  MoveC 2623 to (57.81, -73.19, -4) mm, rotated rx 180 ry 0 rz 90 deg; joints [72.07, -16.046, 78.681, 0, 27.365, 72.07] to (57.8, -69.17, -4) mm, rotated rx 180 ry 0 rz 90 deg; joints [72.193, -16.074, 78.779, 0, 27.295, 72.193]
  MoveL 2624 to (57.48, -68.7, -4) mm, rotated rx -180 ry 0 rz 90 deg; joints [72.204, -16.085, 78.814, 0, 27.271, 72.204]
  MoveL 2625 to (54.49, -65.17, -4) mm, rotated rx 180 ry 0 rz 90 deg; joints [72.283, -16.175, 79.122, 0, 27.052, 72.283]
  MoveL 2626 to (28.89, -35.54, -4) mm, rotated rx -180 ry 0 rz 90 deg; joints [72.956, -16.906, 81.694, 0, 25.212, 72.956]
  MoveL 2627 to (27.54, -34.02, -4) mm, rotated rx 180 ry 0 rz 90 deg; joints [72.991, -16.943, 81.826, 0, 25.117, 72.991]
  MoveL 2628 to (13.23, -22.57, -4) mm, rotated rx 180 ry 0 rz 90 deg; joints [73.216, -17.293, 83.111, 0, 24.182, 73.216]
  MoveC 2629 to (12.1, -21.76, -4) mm, rotated rx -180 ry 0 rz 90 deg; joints [73.231, -17.319, 83.209, 0, 24.11, 73.231] to (10.9, -21.09, -4) mm, rotated rx 180 ry 0 rz 90 deg; joints [73.241, -17.346, 83.31, 0, 24.036, 73.241]
  MoveC 2630 to (6.62, -20.99, -4) mm, rotated rx 180 ry 0 rz 90 deg; joints [73.203, -17.429, 83.618, 0, 23.81, 73.203] to (3.75, -24.17, -4) mm, rotated rx 180 ry 0 rz 90 deg; joints [73.074, -17.465, 83.754, 0, 23.711, 73.074]
  MoveL 2631 to (3.46, -25.11, -4) mm, rotated rx -180 ry 0 rz 90 deg; joints [73.04, -17.465, 83.754, 0, 23.711, 73.04]
  MoveL 2632 to (-7.61, -66.81, -4) mm, rotated rx 180 ry 0 rz 90 deg; joints [71.6, -17.423, 83.597, 0, 23.826, 71.6]
  MoveL 2633 to (-8.62, -70.6, -4) mm, rotated rx 180 ry 0 rz 90 deg; joints [71.469, -17.418, 83.578, 0, 23.84, 71.469]
  MoveL 2634 to (-8.77, -71.55, -4) mm, rotated rx -180 ry 0 rz 90 deg; joints [71.437, -17.415, 83.566, 0, 23.849, 71.437]
  MoveC 2635 to (-8.03, -75.01, -4) mm, rotated rx 180 ry 0 rz 90 deg; joints [71.336, -17.379, 83.432, 0, 23.947, 71.336] to (-5.21, -77.15, -4) mm, rotated rx 180 ry 0 rz 90 deg; joints [71.298, -17.312, 83.181, 0, 24.131, 71.298]
  MoveC 2636 to (-3.81, -77.46, -4) mm, rotated rx -180 ry 0 rz 90 deg; joints [71.303, -17.283, 83.073, 0, 24.21, 71.303] to (-2.37, -77.54, -4) mm, rotated rx -180 ry 0 rz 90 deg; joints [71.316, -17.255, 82.969, 0, 24.286, 71.316]
  MoveL 2637 to (25.78, -77.25, -4) mm, rotated rx 180 ry 0 rz 90 deg; joints [71.62, -16.698, 80.95, 0, 25.748, 71.62]
  MoveL 2638 to (25.7, -69.7, -4) mm, rotated rx 180 ry 0 rz 90 deg; joints [71.855, -16.751, 81.137, 0, 25.614, 71.855]
  MoveL 2639 to (25.7, -69.7, -1) mm, rotated rx 180 ry 0 rz 90 deg; joints [71.855, -16.902, 81.239, 0, 25.664, 71.855]
  Establecer velocidad (1000.0 mm/s)
  MoveL 2640 to (25.7, -69.7, 10) mm, rotated rx 180 ry 0 rz 90 deg; joints [71.855, -17.457, 81.607, 0, 25.851, 71.855]
  Establecer velocidad (66.7 mm/s)
  MoveL 2641 to (67.55, -30.93, 10) mm, rotated rx -180 ry 0 rz 90 deg; joints [73.464, -16.821, 79.406, 0, 27.415, 73.464]
  MoveL 2642 to (67.55, -30.93, -0.75) mm, rotated rx -180 ry 0 rz 90 deg; joints [73.464, -16.283, 79.045, 0, 27.238, 73.464]
  MoveL 2643 to (69.05, -31.11, -1.16) mm, rotated rx -180 ry 0 rz 90 deg; joints [73.472, -16.228, 78.914, 0, 27.314, 73.472]
  MoveL 2644 to (70.56, -30.93, -1.56) mm, rotated rx 180 ry 0 rz 90 deg; joints [73.492, -16.176, 78.79, 0, 27.385, 73.492]
  MoveL 2645 to (71.99, -30.42, -1.97) mm, rotated rx -180 ry 0 rz 90 deg; joints [73.521, -16.127, 78.68, 0, 27.447, 73.521]
  MoveL 2646 to (73.27, -29.6, -2.37) mm, rotated rx 180 ry 0 rz 90 deg; joints [73.558, -16.083, 78.587, 0, 27.496, 73.558]
  MoveL 2647 to (74.34, -28.52, -2.78) mm, rotated rx -180 ry 0 rz 90 deg; joints [73.601, -16.046, 78.516, 0, 27.53, 73.601]
  MoveL 2648 to (75.15, -27.24, -3.19) mm, rotated rx 180 ry 0 rz 90 deg; joints [73.648, -16.016, 78.47, 0, 27.546, 73.648]
  MoveL 2649 to (75.65, -25.8, -3.59) mm, rotated rx -180 ry 0 rz 90 deg; joints [73.696, -15.994, 78.45, 0, 27.544, 73.696]
  MoveL 2650 to (75.78, -24.29, -4) mm, rotated rx -180 ry 0 rz 90 deg; joints [73.744, -15.98, 78.46, 0, 27.521, 73.744]
  MoveL 2651 to (75.78, -5.21, -4) mm, rotated rx -180 ry 0 rz 90 deg; joints [74.335, -16.102, 78.873, 0, 27.229, 74.335]
  MoveL 2652 to (75.77, -4.51, -4) mm, rotated rx 180 ry 0 rz 90 deg; joints [74.357, -16.107, 78.889, 0, 27.217, 74.357]
  MoveC 2653 to (73.31, -1.48, -4) mm, rotated rx -180 ry 0 rz 90 deg; joints [74.43, -16.18, 79.139, 0, 27.041, 74.43] to (69.65, -0.12, -4) mm, rotated rx -180 ry 0 rz 90 deg; joints [74.44, -16.268, 79.443, 0, 26.825, 74.44]
  MoveC 2654 to (68.39, -0.22, -4) mm, rotated rx 180 ry 0 rz 90 deg; joints [74.426, -16.295, 79.536, 0, 26.759, 74.426] to (67.21, -0.66, -4) mm, rotated rx -180 ry 0 rz 90 deg; joints [74.402, -16.318, 79.615, 0, 26.702, 74.402]
  MoveL 2655 to (66.63, -1.42, -4) mm, rotated rx 180 ry 0 rz 90 deg; joints [74.373, -16.326, 79.643, 0, 26.683, 74.373]
  MoveL 2656 to (51.65, -21.98, -4) mm, rotated rx 180 ry 0 rz 90 deg; joints [73.596, -16.52, 80.321, 0, 26.199, 73.596]
  MoveL 2657 to (50.74, -23.24, -4) mm, rotated rx 180 ry 0 rz 90 deg; joints [73.549, -16.531, 80.36, 0, 26.171, 73.549]
  MoveC 2658 to (49.85, -26.2, -4) mm, rotated rx 180 ry 0 rz 90 deg; joints [73.448, -16.532, 80.361, 0, 26.17, 73.448] to (50.96, -29.09, -4) mm, rotated rx -180 ry 0 rz 90 deg; joints [73.368, -16.49, 80.215, 0, 26.275, 73.368]
  MoveL 2659 to (51.59, -29.85, -4) mm, rotated rx -180 ry 0 rz 90 deg; joints [73.35, -16.472, 80.151, 0, 26.32, 73.35]
  MoveL 2660 to (67.24, -47.54, -4) mm, rotated rx 180 ry 0 rz 90 deg; joints [72.949, -16.016, 78.579, 0, 27.436, 72.949]
  MoveL 2661 to (67.55, -47.86, -4) mm, rotated rx -180 ry 0 rz 90 deg; joints [72.942, -16.007, 78.549, 0, 27.458, 72.942]
  MoveC 2662 to (68.55, -48.33, -4) mm, rotated rx -180 ry 0 rz 90 deg; joints [72.937, -15.981, 78.463, 0, 27.519, 72.937] to (69.65, -48.44, -4) mm, rotated rx -180 ry 0 rz 90 deg; joints [72.944, -15.956, 78.377, 0, 27.579, 72.944]
  MoveC 2663 to (73.34, -47.15, -4) mm, rotated rx 180 ry 0 rz 90 deg; joints [73.018, -15.882, 78.127, 0, 27.755, 73.018] to (75.75, -44.07, -4) mm, rotated rx -180 ry 0 rz 90 deg; joints [73.135, -15.849, 78.016, 0, 27.833, 73.135]
  MoveL 2664 to (75.79, -43.12, -4) mm, rotated rx 180 ry 0 rz 90 deg; joints [73.165, -15.855, 78.034, 0, 27.82, 73.165]
  MoveL 2665 to (75.78, -24.29, -4) mm, rotated rx -180 ry 0 rz 90 deg; joints [73.744, -15.98, 78.46, 0, 27.521, 73.744]
  MoveL 2666 to (68.23, -24.29, -4) mm, rotated rx 180 ry 0 rz 90 deg; joints [73.676, -16.148, 79.03, 0, 27.118, 73.676]
  MoveL 2667 to (68.23, -24.29, -1) mm, rotated rx -180 ry 0 rz 90 deg; joints [73.676, -16.298, 79.132, 0, 27.166, 73.676]
  Establecer velocidad (1000.0 mm/s)
  MoveL 2668 to (68.23, -24.29, 10) mm, rotated rx 180 ry 0 rz 90 deg; joints [73.676, -16.849, 79.502, 0, 27.348, 73.676]
  Establecer velocidad (66.7 mm/s)
  MoveL 2669 to (36.34, 8.62, 10) mm, rotated rx 180 ry 0 rz 90 deg; joints [74.423, -17.725, 82.561, 0, 25.164, 74.423]
  MoveL 2670 to (36.34, 8.62, -0.75) mm, rotated rx 180 ry 0 rz 90 deg; joints [74.423, -17.181, 82.202, 0, 24.979, 74.423]
  MoveL 2671 to (37.46, 7.59, -1.16) mm, rotated rx 180 ry 0 rz 90 deg; joints [74.4, -17.132, 82.086, 0, 25.046, 74.4]
  MoveL 2672 to (38.79, 6.86, -1.56) mm, rotated rx -180 ry 0 rz 90 deg; joints [74.389, -17.08, 81.96, 0, 25.12, 74.389]
  MoveL 2673 to (40.25, 6.44, -1.97) mm, rotated rx 180 ry 0 rz 90 deg; joints [74.389, -17.028, 81.831, 0, 25.197, 74.389]
  MoveL 2674 to (41.77, 6.36, -2.37) mm, rotated rx -180 ry 0 rz 90 deg; joints [74.399, -16.976, 81.704, 0, 25.272, 74.399]
  MoveL 2675 to (43.27, 6.61, -2.78) mm, rotated rx 180 ry 0 rz 90 deg; joints [74.421, -16.926, 81.585, 0, 25.341, 74.421]
  MoveL 2676 to (44.68, 7.19, -3.19) mm, rotated rx 180 ry 0 rz 90 deg; joints [74.452, -16.88, 81.48, 0, 25.4, 74.452]
  MoveL 2677 to (45.92, 8.07, -3.59) mm, rotated rx 180 ry 0 rz 90 deg; joints [74.49, -16.839, 81.393, 0, 25.446, 74.49]
  MoveL 2678 to (46.91, 9.21, -4) mm, rotated rx 180 ry 0 rz 90 deg; joints [74.535, -16.805, 81.329, 0, 25.475, 74.535]
  MoveL 2679 to (58.63, 25.57, -4) mm, rotated rx 180 ry 0 rz 90 deg; joints [75.153, -16.653, 80.79, 0, 25.864, 75.153]
  MoveC 2680 to (58.89, 26.03, -4) mm, rotated rx 180 ry 0 rz 90 deg; joints [75.17, -16.65, 80.779, 0, 25.871, 75.17] to (59.04, 26.54, -4) mm, rotated rx 180 ry 0 rz 90 deg; joints [75.187, -16.65, 80.778, 0, 25.872, 75.187]
  MoveC 2681 to (58.64, 30.12, -4) mm, rotated rx 180 ry 0 rz 90 deg; joints [75.297, -16.678, 80.878, 0, 25.8, 75.297] to (56.35, 32.91, -4) mm, rotated rx -180 ry 0 rz 90 deg; joints [75.366, -16.741, 81.102, 0, 25.639, 75.366]
  MoveC 2682 to (55.39, 33.36, -4) mm, rotated rx -180 ry 0 rz 90 deg; joints [75.373, -16.764, 81.183, 0, 25.581, 75.373] to (54.33, 33.5, -4) mm, rotated rx -180 ry 0 rz 90 deg; joints [75.368, -16.786, 81.264, 0, 25.523, 75.368]
  MoveL 2683 to (46.91, 33.32, -4) mm, rotated rx -180 ry 0 rz 90 deg; joints [75.301, -16.938, 81.808, 0, 25.13, 75.301]
  MoveL 2684 to (7.5, 32.25, -4) mm, rotated rx 180 ry 0 rz 90 deg; joints [74.929, -17.696, 84.638, 0, 23.058, 74.929]
  MoveC 2685 to (4.94, 31.58, -4) mm, rotated rx -180 ry 0 rz 90 deg; joints [74.885, -17.74, 84.808, 0, 22.932, 74.885] to (2.93, 29.85, -4) mm, rotated rx -180 ry 0 rz 90 deg; joints [74.811, -17.768, 84.917, 0, 22.852, 74.811]
  MoveC 2686 to (2.15, 27.7, -4) mm, rotated rx 180 ry 0 rz 90 deg; joints [74.734, -17.772, 84.931, 0, 22.841, 74.734] to (2.37, 25.41, -4) mm, rotated rx -180 ry 0 rz 90 deg; joints [74.661, -17.757, 84.871, 0, 22.886, 74.661]
  MoveL 2687 to (2.79, 24.17, -4) mm, rotated rx -180 ry 0 rz 90 deg; joints [74.625, -17.743, 84.817, 0, 22.926, 74.625]
  MoveL 2688 to (8.64, 8.05, -4) mm, rotated rx -180 ry 0 rz 90 deg; joints [74.155, -17.551, 84.08, 0, 23.47, 74.155]
  MoveC 2689 to (9.35, 6.7, -4) mm, rotated rx -180 ry 0 rz 90 deg; joints [74.118, -17.53, 84.002, 0, 23.528, 74.118] to (10.39, 5.59, -4) mm, rotated rx 180 ry 0 rz 90 deg; joints [74.092, -17.505, 83.906, 0, 23.599, 74.092]
  MoveL 2690 to (27.01, -7.35, -4) mm, rotated rx 180 ry 0 rz 90 deg; joints [73.831, -17.112, 82.441, 0, 24.67, 73.831]
  MoveL 2691 to (27.96, -8.06, -4) mm, rotated rx -180 ry 0 rz 90 deg; joints [73.817, -17.089, 82.358, 0, 24.731, 73.817]
  MoveC 2692 to (31.75, -9.06, -4) mm, rotated rx -180 ry 0 rz 90 deg; joints [73.82, -17.007, 82.061, 0, 24.946, 73.82] to (35.15, -7.11, -4) mm, rotated rx 180 ry 0 rz 90 deg; joints [73.913, -16.95, 81.854, 0, 25.096, 73.913]
  MoveL 2693 to (35.89, -6.16, -4) mm, rotated rx 180 ry 0 rz 90 deg; joints [73.95, -16.941, 81.82, 0, 25.121, 73.95]
  MoveL 2694 to (46.91, 9.21, -4) mm, rotated rx 180 ry 0 rz 90 deg; joints [74.535, -16.805, 81.329, 0, 25.475, 74.535]
  MoveL 2695 to (40.77, 13.61, -4) mm, rotated rx -180 ry 0 rz 90 deg; joints [74.621, -16.955, 81.87, 0, 25.085, 74.621]
  MoveL 2696 to (40.77, 13.61, -1) mm, rotated rx 180 ry 0 rz 90 deg; joints [74.621, -17.107, 81.971, 0, 25.136, 74.621]
  Establecer velocidad (1000.0 mm/s)
  MoveL 2697 to (40.77, 13.61, 10) mm, rotated rx 180 ry 0 rz 90 deg; joints [74.621, -17.663, 82.338, 0, 25.325, 74.621]
  Establecer velocidad (66.7 mm/s)
  MoveL 2698 to (26.76, 68.82, 10) mm, rotated rx -180 ry 0 rz 90 deg; joints [76.28, -18.225, 84.399, 0, 23.827, 76.28]
  MoveL 2699 to (26.76, 68.82, -0.75) mm, rotated rx -180 ry 0 rz 90 deg; joints [76.28, -17.677, 84.041, 0, 23.637, 76.28]
  MoveL 2700 to (26.96, 70.32, -1.16) mm, rotated rx 180 ry 0 rz 90 deg; joints [76.331, -17.66, 84.039, 0, 23.621, 76.331]
  MoveL 2701 to (26.79, 71.84, -1.56) mm, rotated rx 180 ry 0 rz 90 deg; joints [76.379, -17.649, 84.064, 0, 23.585, 76.379]
  MoveL 2702 to (26.29, 73.27, -1.97) mm, rotated rx 180 ry 0 rz 90 deg; joints [76.422, -17.645, 84.111, 0, 23.534, 76.422]
  MoveL 2703 to (25.49, 74.56, -2.37) mm, rotated rx 180 ry 0 rz 90 deg; joints [76.457, -17.645, 84.177, 0, 23.467, 76.457]
  MoveL 2704 to (24.42, 75.64, -2.78) mm, rotated rx 180 ry 0 rz 90 deg; joints [76.484, -17.649, 84.259, 0, 23.39, 76.484]
  MoveL 2705 to (23.14, 76.46, -3.19) mm, rotated rx 180 ry 0 rz 90 deg; joints [76.501, -17.656, 84.352, 0, 23.304, 76.501]
  MoveL 2706 to (21.71, 76.98, -3.59) mm, rotated rx -180 ry 0 rz 90 deg; joints [76.506, -17.665, 84.45, 0, 23.215, 76.506]
  MoveL 2707 to (20.21, 77.13, -4) mm, rotated rx -180 ry 0 rz 90 deg; joints [76.5, -17.673, 84.547, 0, 23.126, 76.5]
  MoveL 2708 to (-28.9, 77.66, -4) mm, rotated rx -180 ry 0 rz 90 deg; joints [76.12, -18.533, 88.011, 0, 20.522, 76.12]
  MoveL 2709 to (-30.61, 77.66, -4) mm, rotated rx -180 ry 0 rz 90 deg; joints [76.106, -18.561, 88.129, 0, 20.432, 76.106]
  MoveC 2710 to (-32.6, 77.56, -4) mm, rotated rx -180 ry 0 rz 90 deg; joints [76.086, -18.593, 88.264, 0, 20.329, 76.086] to (-34.56, 77.23, -4) mm, rotated rx 180 ry 0 rz 90 deg; joints [76.059, -18.623, 88.394, 0, 20.23, 76.059]
  MoveC 2711 to (-37.55, 73.36, -4) mm, rotated rx 180 ry 0 rz 90 deg; joints [75.903, -18.656, 88.533, 0, 20.123, 75.903] to (-36.68, 68.53, -4) mm, rotated rx 180 ry 0 rz 90 deg; joints [75.748, -18.622, 88.389, 0, 20.233, 75.748]
  MoveC 2712 to (-34.85, 67.27, -4) mm, rotated rx 180 ry 0 rz 90 deg; joints [75.721, -18.588, 88.242, 0, 20.346, 75.721] to (-32.99, 66.06, -4) mm, rotated rx -180 ry 0 rz 90 deg; joints [75.696, -18.553, 88.092, 0, 20.46, 75.696]
  MoveL 2713 to (-12.79, 53.26, -4) mm, rotated rx 180 ry 0 rz 90 deg; joints [75.443, -18.159, 86.463, 0, 21.696, 75.443]
  MoveL 2714 to (-11.85, 52.68, -4) mm, rotated rx 180 ry 0 rz 90 deg; joints [75.431, -18.14, 86.386, 0, 21.754, 75.431]
  MoveC 2715 to (-9.56, 51.76, -4) mm, rotated rx -180 ry 0 rz 90 deg; joints [75.421, -18.096, 86.209, 0, 21.887, 75.421] to (-7.11, 51.53, -4) mm, rotated rx -180 ry 0 rz 90 deg; joints [75.434, -18.052, 86.032, 0, 22.019, 75.434]
  MoveL 2716 to (70.6, 57.18, -4) mm, rotated rx 180 ry 0 rz 90 deg; joints [76.25, -16.57, 80.498, 0, 26.073, 76.25]
  MoveL 2717 to (71.37, 57.27, -4) mm, rotated rx 180 ry 0 rz 90 deg; joints [76.259, -16.554, 80.441, 0, 26.113, 76.259]
  MoveC 2718 to (74.16, 58.71, -4) mm, rotated rx 180 ry 0 rz 90 deg; joints [76.327, -16.502, 80.258, 0, 26.244, 76.327] to (75.32, 61.63, -4) mm, rotated rx -180 ry 0 rz 90 deg; joints [76.428, -16.493, 80.225, 0, 26.268, 76.428]
  MoveL 2719 to (75.32, 62.07, -4) mm, rotated rx 180 ry 0 rz 90 deg; joints [76.442, -16.495, 80.232, 0, 26.263, 76.442]
  MoveL 2720 to (75.32, 71.55, -4) mm, rotated rx -180 ry 0 rz 90 deg; joints [76.742, -16.543, 80.402, 0, 26.141, 76.742]
  MoveL 2721 to (75.31, 71.95, -4) mm, rotated rx -180 ry 0 rz 90 deg; joints [76.755, -16.546, 80.411, 0, 26.135, 76.755]
  MoveC 2722 to (74, 74.91, -4) mm, rotated rx 180 ry 0 rz 90 deg; joints [76.839, -16.588, 80.561, 0, 26.027, 76.839] to (71.02, 76.18, -4) mm, rotated rx -180 ry 0 rz 90 deg; joints [76.858, -16.658, 80.807, 0, 25.851, 76.858]
  MoveC 2723 to (46.95, 76.74, -4) mm, rotated rx 180 ry 0 rz 90 deg; joints [76.694, -17.155, 82.6, 0, 24.555, 76.694] to (22.88, 77.1, -4) mm, rotated rx -180 ry 0 rz 90 deg; joints [76.52, -17.623, 84.355, 0, 23.268, 76.52]
  MoveL 2724 to (20.21, 77.13, -4) mm, rotated rx -180 ry 0 rz 90 deg; joints [76.5, -17.673, 84.547, 0, 23.126, 76.5]
  MoveL 2725 to (20.12, 69.58, -4) mm, rotated rx -180 ry 0 rz 90 deg; joints [76.252, -17.64, 84.422, 0, 23.218, 76.252]
  MoveL 2726 to (20.12, 69.58, -1) mm, rotated rx 180 ry 0 rz 90 deg; joints [76.252, -17.793, 84.523, 0, 23.271, 76.252]
  Establecer velocidad (1000.0 mm/s)
  MoveL 2727 to (20.12, 69.58, 10) mm, rotated rx -180 ry 0 rz 90 deg; joints [76.252, -18.355, 84.889, 0, 23.466, 76.252]
  Establecer velocidad (66.7 mm/s)
  MoveL 2728 to (26.76, 68.55, 10) mm, rotated rx 180 ry 0 rz 90 deg; joints [76.271, -18.224, 84.394, 0, 23.83, 76.271]
  MoveL 2729 to (26.76, 68.55, -1) mm, rotated rx -180 ry 0 rz 90 deg; joints [76.271, -17.663, 84.027, 0, 23.636, 76.271]
  MoveL 2730 to (26.96, 70.05, -1.41) mm, rotated rx 180 ry 0 rz 90 deg; joints [76.322, -17.646, 84.026, 0, 23.62, 76.322]
  MoveL 2731 to (26.79, 71.56, -1.81) mm, rotated rx 180 ry 0 rz 90 deg; joints [76.37, -17.635, 84.05, 0, 23.585, 76.37]
  MoveL 2732 to (26.29, 73, -2.22) mm, rotated rx 180 ry 0 rz 90 deg; joints [76.413, -17.63, 84.098, 0, 23.533, 76.413]
  MoveL 2733 to (25.49, 74.29, -2.62) mm, rotated rx 180 ry 0 rz 90 deg; joints [76.448, -17.631, 84.164, 0, 23.467, 76.448]
  MoveL 2734 to (24.42, 75.37, -3.03) mm, rotated rx -180 ry 0 rz 90 deg; joints [76.475, -17.635, 84.247, 0, 23.389, 76.475]
  MoveL 2735 to (23.14, 76.19, -3.44) mm, rotated rx 180 ry 0 rz 90 deg; joints [76.492, -17.642, 84.339, 0, 23.303, 76.492]
  MoveL 2736 to (21.71, 76.7, -3.84) mm, rotated rx 180 ry 0 rz 90 deg; joints [76.497, -17.651, 84.437, 0, 23.214, 76.497]
  MoveL 2737 to (20.2, 76.86, -4.25) mm, rotated rx 180 ry 0 rz 90 deg; joints [76.491, -17.659, 84.534, 0, 23.125, 76.491]
  MoveC 2738 to (19.81, 76.86, -4.25) mm, rotated rx 180 ry 0 rz 90 deg; joints [76.488, -17.666, 84.562, 0, 23.104, 76.488] to (19.43, 76.86, -4.25) mm, rotated rx -180 ry 0 rz 90 deg; joints [76.485, -17.673, 84.59, 0, 23.083, 76.485]
  MoveL 2739 to (-29.85, 77.36, -4.25) mm, rotated rx -180 ry 0 rz 90 deg; joints [76.102, -18.535, 88.063, 0, 20.472, 76.102]
  MoveC 2740 to (-31.85, 77.3, -4.25) mm, rotated rx -180 ry 0 rz 90 deg; joints [76.084, -18.567, 88.2, 0, 20.367, 76.084] to (-33.83, 77.08, -4.25) mm, rotated rx 180 ry 0 rz 90 deg; joints [76.06, -18.598, 88.333, 0, 20.266, 76.06]
  MoveC 2741 to (-36.86, 73.32, -4.25) mm, rotated rx -180 ry 0 rz 90 deg; joints [75.907, -18.632, 88.476, 0, 20.156, 75.907] to (-36.19, 68.55, -4.25) mm, rotated rx 180 ry 0 rz 90 deg; joints [75.752, -18.602, 88.347, 0, 20.254, 75.752]
  MoveL 2742 to (-34.59, 67.43, -4.25) mm, rotated rx 180 ry 0 rz 90 deg; joints [75.728, -18.571, 88.218, 0, 20.353, 75.728]
  MoveL 2743 to (-27.63, 63.02, -4.25) mm, rotated rx -180 ry 0 rz 90 deg; joints [75.64, -18.439, 87.661, 0, 20.778, 75.64]
  MoveL 2744 to (-11.99, 53.11, -4.25) mm, rotated rx 180 ry 0 rz 90 deg; joints [75.444, -18.131, 86.395, 0, 21.736, 75.444]
  MoveC 2745 to (-9.54, 52.06, -4.25) mm, rotated rx 180 ry 0 rz 90 deg; joints [75.431, -18.084, 86.204, 0, 21.88, 75.431] to (-6.89, 51.83, -4.25) mm, rotated rx 180 ry 0 rz 90 deg; joints [75.446, -18.036, 86.014, 0, 22.022, 75.446]
  MoveC 2746 to (28.54, 54.43, -4.25) mm, rotated rx 180 ry 0 rz 90 deg; joints [75.827, -17.396, 83.536, 0, 23.86, 75.827] to (63.97, 57, -4.25) mm, rotated rx 180 ry 0 rz 90 deg; joints [76.193, -16.697, 80.982, 0, 25.715, 76.193]
  MoveL 2747 to (70.93, 57.56, -4.25) mm, rotated rx 180 ry 0 rz 90 deg; joints [76.265, -16.553, 80.471, 0, 26.082, 76.265]
  MoveC 2748 to (73.83, 58.97, -4.25) mm, rotated rx 180 ry 0 rz 90 deg; joints [76.332, -16.498, 80.28, 0, 26.219, 76.332] to (75, 61.98, -4.25) mm, rotated rx -180 ry 0 rz 90 deg; joints [76.436, -16.489, 80.246, 0, 26.243, 76.436]
  MoveL 2749 to (75, 71.52, -4.25) mm, rotated rx -180 ry 0 rz 90 deg; joints [76.739, -16.537, 80.417, 0, 26.12, 76.739]
  MoveC 2750 to (73.78, 74.54, -4.25) mm, rotated rx -180 ry 0 rz 90 deg; joints [76.826, -16.579, 80.563, 0, 26.016, 76.826] to (70.79, 75.86, -4.25) mm, rotated rx -180 ry 0 rz 90 deg; joints [76.845, -16.649, 80.81, 0, 25.839, 76.845]
  MoveC 2751 to (45.5, 76.48, -4.25) mm, rotated rx -180 ry 0 rz 90 deg; joints [76.674, -17.17, 82.694, 0, 24.476, 76.674] to (20.2, 76.86, -4.25) mm, rotated rx 180 ry 0 rz 90 deg; joints [76.491, -17.659, 84.534, 0, 23.125, 76.491]
  MoveL 2752 to (20.12, 69.31, -4.25) mm, rotated rx -180 ry 0 rz 90 deg; joints [76.243, -17.626, 84.409, 0, 23.218, 76.243]
  MoveL 2753 to (20.12, 69.31, -1.25) mm, rotated rx 180 ry 0 rz 90 deg; joints [76.243, -17.779, 84.51, 0, 23.27, 76.243]
  Establecer velocidad (1000.0 mm/s)
  MoveL 2754 to (20.12, 69.31, 10) mm, rotated rx 180 ry 0 rz 90 deg; joints [76.243, -18.354, 84.884, 0, 23.47, 76.243]
  Establecer velocidad (66.7 mm/s)
  MoveL 2755 to (37.85, 24.53, 10) mm, rotated rx 180 ry 0 rz 90 deg; joints [74.944, -17.783, 82.769, 0, 25.013, 74.944]
  MoveL 2756 to (37.85, 24.53, -1) mm, rotated rx -180 ry 0 rz 90 deg; joints [74.944, -17.225, 82.402, 0, 24.823, 74.944]
  MoveL 2757 to (38, 26.04, -1.41) mm, rotated rx 180 ry 0 rz 90 deg; joints [74.993, -17.21, 82.407, 0, 24.803, 74.993]
  MoveL 2758 to (37.77, 27.54, -1.81) mm, rotated rx 180 ry 0 rz 90 deg; joints [75.039, -17.202, 82.439, 0, 24.763, 75.039]
  MoveL 2759 to (37.22, 28.96, -2.22) mm, rotated rx 180 ry 0 rz 90 deg; joints [75.08, -17.2, 82.493, 0, 24.706, 75.08]
  MoveL 2760 to (36.37, 30.22, -2.62) mm, rotated rx -180 ry 0 rz 90 deg; joints [75.113, -17.203, 82.566, 0, 24.637, 75.113]
  MoveL 2761 to (35.26, 31.26, -3.03) mm, rotated rx -180 ry 0 rz 90 deg; joints [75.137, -17.21, 82.653, 0, 24.556, 75.137]
  MoveL 2762 to (33.95, 32.03, -3.44) mm, rotated rx 180 ry 0 rz 90 deg; joints [75.15, -17.219, 82.75, 0, 24.469, 75.15]
  MoveL 2763 to (32.5, 32.49, -3.84) mm, rotated rx -180 ry 0 rz 90 deg; joints [75.153, -17.229, 82.85, 0, 24.379, 75.153]
  MoveL 2764 to (30.99, 32.59, -4.25) mm, rotated rx 180 ry 0 rz 90 deg; joints [75.143, -17.239, 82.948, 0, 24.29, 75.143]
  MoveL 2765 to (8.05, 31.96, -4.25) mm, rotated rx 180 ry 0 rz 90 deg; joints [74.925, -17.672, 84.585, 0, 23.087, 74.925]
  MoveL 2766 to (7.11, 31.9, -4.25) mm, rotated rx 180 ry 0 rz 90 deg; joints [74.914, -17.689, 84.651, 0, 23.038, 74.914]
  MoveC 2767 to (3.22, 29.6, -4.25) mm, rotated rx -180 ry 0 rz 90 deg; joints [74.805, -17.749, 84.884, 0, 22.866, 74.805] to (2.78, 25.11, -4.25) mm, rotated rx 180 ry 0 rz 90 deg; joints [74.655, -17.735, 84.828, 0, 22.907, 74.655]
  MoveL 2768 to (8.98, 8.05, -4.25) mm, rotated rx -180 ry 0 rz 90 deg; joints [74.159, -17.532, 84.048, 0, 23.484, 74.159]
  MoveC 2769 to (9.63, 6.82, -4.25) mm, rotated rx 180 ry 0 rz 90 deg; joints [74.125, -17.513, 83.977, 0, 23.536, 74.125] to (10.59, 5.81, -4.25) mm, rotated rx -180 ry 0 rz 90 deg; joints [74.101, -17.489, 83.887, 0, 23.602, 74.101]
  MoveL 2770 to (28.01, -7.75, -4.25) mm, rotated rx -180 ry 0 rz 90 deg; joints [73.827, -17.077, 82.352, 0, 24.725, 73.827]
  MoveC 2771 to (31.6, -8.76, -4.25) mm, rotated rx -180 ry 0 rz 90 deg; joints [73.828, -17, 82.07, 0, 24.93, 73.828] to (34.86, -6.95, -4.25) mm, rotated rx 180 ry 0 rz 90 deg; joints [73.915, -16.944, 81.87, 0, 25.075, 73.915]
  MoveL 2772 to (35.5, -6.16, -4.25) mm, rotated rx -180 ry 0 rz 90 deg; joints [73.946, -16.936, 81.84, 0, 25.097, 73.946]
  MoveL 2773 to (40.27, 0.5, -4.25) mm, rotated rx -180 ry 0 rz 90 deg; joints [74.201, -16.878, 81.63, 0, 25.248, 74.201]
  MoveL 2774 to (40.95, 1.42, -4.25) mm, rotated rx -180 ry 0 rz 90 deg; joints [74.236, -16.869, 81.599, 0, 25.271, 74.236]
  MoveL 2775 to (57.96, 25.11, -4.25) mm, rotated rx 180 ry 0 rz 90 deg; joints [75.133, -16.652, 80.823, 0, 25.83, 75.133]
  MoveL 2776 to (58.35, 25.73, -4.25) mm, rotated rx -180 ry 0 rz 90 deg; joints [75.156, -16.647, 80.805, 0, 25.842, 75.156]
  MoveC 2777 to (58.06, 30.12, -4.25) mm, rotated rx 180 ry 0 rz 90 deg; joints [75.292, -16.678, 80.913, 0, 25.765, 75.292] to (54.87, 33.14, -4.25) mm, rotated rx 180 ry 0 rz 90 deg; joints [75.362, -16.761, 81.208, 0, 25.552, 75.362]
  MoveL 2778 to (54.49, 33.2, -4.25) mm, rotated rx -180 ry 0 rz 90 deg; joints [75.36, -16.769, 81.238, 0, 25.531, 75.36]
  MoveL 2779 to (50.7, 33.12, -4.25) mm, rotated rx 180 ry 0 rz 90 deg; joints [75.326, -16.847, 81.516, 0, 25.33, 75.326]
  MoveL 2780 to (30.99, 32.59, -4.25) mm, rotated rx 180 ry 0 rz 90 deg; joints [75.143, -17.239, 82.948, 0, 24.29, 75.143]
  MoveL 2781 to (31.2, 25.04, -4.25) mm, rotated rx 180 ry 0 rz 90 deg; joints [74.903, -17.195, 82.787, 0, 24.408, 74.903]
  MoveL 2782 to (31.2, 25.04, -1.25) mm, rotated rx 180 ry 0 rz 90 deg; joints [74.903, -17.348, 82.888, 0, 24.459, 74.903]
  Establecer velocidad (1000.0 mm/s)
  MoveL 2783 to (31.2, 25.04, 10) mm, rotated rx 180 ry 0 rz 90 deg; joints [74.903, -17.919, 83.263, 0, 24.655, 74.903]
  Establecer velocidad (66.7 mm/s)
  MoveL 2784 to (67.24, -30.95, 10) mm, rotated rx -180 ry 0 rz 90 deg; joints [73.461, -16.828, 79.428, 0, 27.399, 73.461]
  MoveL 2785 to (67.24, -30.95, -1) mm, rotated rx 180 ry 0 rz 90 deg; joints [73.461, -16.277, 79.059, 0, 27.218, 73.461]
  MoveL 2786 to (68.75, -31.14, -1.41) mm, rotated rx 180 ry 0 rz 90 deg; joints [73.469, -16.222, 78.928, 0, 27.295, 73.469]
  MoveL 2787 to (70.26, -30.95, -1.81) mm, rotated rx 180 ry 0 rz 90 deg; joints [73.488, -16.17, 78.804, 0, 27.365, 73.488]
  MoveL 2788 to (71.69, -30.44, -2.22) mm, rotated rx 180 ry 0 rz 90 deg; joints [73.517, -16.121, 78.693, 0, 27.427, 73.517]
  MoveL 2789 to (72.97, -29.62, -2.62) mm, rotated rx 180 ry 0 rz 90 deg; joints [73.554, -16.077, 78.601, 0, 27.476, 73.554]
  MoveL 2790 to (74.04, -28.54, -3.03) mm, rotated rx 180 ry 0 rz 90 deg; joints [73.597, -16.04, 78.53, 0, 27.51, 73.597]
  MoveL 2791 to (74.84, -27.26, -3.44) mm, rotated rx -180 ry 0 rz 90 deg; joints [73.644, -16.01, 78.484, 0, 27.526, 73.644]
  MoveL 2792 to (75.34, -25.82, -3.84) mm, rotated rx -180 ry 0 rz 90 deg; joints [73.693, -15.988, 78.464, 0, 27.524, 73.693]
  MoveL 2793 to (75.48, -24.31, -4.25) mm, rotated rx 180 ry 0 rz 90 deg; joints [73.741, -15.975, 78.473, 0, 27.501, 73.741]
  MoveL 2794 to (75.48, -6.16, -4.25) mm, rotated rx -180 ry 0 rz 90 deg; joints [74.303, -16.09, 78.867, 0, 27.223, 74.303]
  MoveL 2795 to (75.47, -5.19, -4.25) mm, rotated rx 180 ry 0 rz 90 deg; joints [74.333, -16.096, 78.888, 0, 27.208, 74.333]
  MoveC 2796 to (73.5, -2.57, -4.25) mm, rotated rx 180 ry 0 rz 90 deg; joints [74.397, -16.156, 79.093, 0, 27.063, 74.397] to (70.6, -1.03, -4.25) mm, rotated rx 180 ry 0 rz 90 deg; joints [74.42, -16.229, 79.344, 0, 26.885, 74.42]
  MoveC 2797 to (68.82, -0.84, -4.25) mm, rotated rx 180 ry 0 rz 90 deg; joints [74.41, -16.269, 79.482, 0, 26.787, 74.41] to (67.09, -1.32, -4.25) mm, rotated rx -180 ry 0 rz 90 deg; joints [74.38, -16.304, 79.602, 0, 26.702, 74.38]
  MoveL 2798 to (65.86, -2.99, -4.25) mm, rotated rx -180 ry 0 rz 90 deg; joints [74.318, -16.32, 79.659, 0, 26.661, 74.318]
  MoveL 2799 to (51.11, -23.22, -4.25) mm, rotated rx -180 ry 0 rz 90 deg; joints [73.553, -16.511, 80.325, 0, 26.186, 73.553]
  MoveC 2800 to (50.17, -26.07, -4.25) mm, rotated rx 180 ry 0 rz 90 deg; joints [73.455, -16.513, 80.332, 0, 26.181, 73.455] to (51.18, -28.9, -4.25) mm, rotated rx 180 ry 0 rz 90 deg; joints [73.376, -16.474, 80.195, 0, 26.279, 73.376]
  MoveL 2801 to (51.65, -29.47, -4.25) mm, rotated rx -180 ry 0 rz 90 deg; joints [73.363, -16.461, 80.148, 0, 26.313, 73.363]
  MoveL 2802 to (67.43, -47.29, -4.25) mm, rotated rx -180 ry 0 rz 90 deg; joints [72.958, -16.001, 78.563, 0, 27.438, 72.958]
  MoveL 2803 to (67.55, -47.4, -4.25) mm, rotated rx 180 ry 0 rz 90 deg; joints [72.956, -15.997, 78.551, 0, 27.446, 72.956]
  MoveC 2804 to (70.08, -47.77, -4.25) mm, rotated rx 180 ry 0 rz 90 deg; joints [72.969, -15.939, 78.351, 0, 27.587, 72.969] to (72.49, -46.9, -4.25) mm, rotated rx 180 ry 0 rz 90 deg; joints [73.018, -15.89, 78.189, 0, 27.702, 73.018]
  MoveL 2805 to (73.09, -46.48, -4.25) mm, rotated rx -180 ry 0 rz 90 deg; joints [73.037, -15.88, 78.153, 0, 27.727, 73.037]
  MoveC 2806 to (74.5, -45.12, -4.25) mm, rotated rx 180 ry 0 rz 90 deg; joints [73.091, -15.857, 78.077, 0, 27.78, 73.091] to (75.47, -43.43, -4.25) mm, rotated rx -180 ry 0 rz 90 deg; joints [73.152, -15.847, 78.043, 0, 27.804, 73.152]
  MoveL 2807 to (75.48, -43.12, -4.25) mm, rotated rx -180 ry 0 rz 90 deg; joints [73.162, -15.849, 78.049, 0, 27.8, 73.162]
  MoveL 2808 to (75.48, -24.31, -4.25) mm, rotated rx 180 ry 0 rz 90 deg; joints [73.741, -15.975, 78.473, 0, 27.501, 73.741]
  MoveL 2809 to (67.93, -24.31, -4.25) mm, rotated rx 180 ry 0 rz 90 deg; joints [73.673, -16.142, 79.044, 0, 27.098, 73.673]
  MoveL 2810 to (67.93, -24.31, -1.25) mm, rotated rx 180 ry 0 rz 90 deg; joints [73.673, -16.292, 79.146, 0, 27.146, 73.673]
  Establecer velocidad (1000.0 mm/s)
  MoveL 2811 to (67.93, -24.31, 10) mm, rotated rx -180 ry 0 rz 90 deg; joints [73.673, -16.856, 79.524, 0, 27.332, 73.673]
  Establecer velocidad (66.7 mm/s)
  MoveL 2812 to (19, -68.78, 10) mm, rotated rx 180 ry 0 rz 90 deg; joints [71.815, -17.6, 82.115, 0, 25.486, 71.815]
  MoveL 2813 to (19, -68.78, -1) mm, rotated rx 180 ry 0 rz 90 deg; joints [71.815, -17.045, 81.747, 0, 25.297, 71.815]
  MoveL 2814 to (18.83, -70.28, -1.41) mm, rotated rx -180 ry 0 rz 90 deg; joints [71.766, -17.017, 81.71, 0, 25.308, 71.766]
  MoveL 2815 to (19.02, -71.79, -1.81) mm, rotated rx 180 ry 0 rz 90 deg; joints [71.721, -16.983, 81.646, 0, 25.337, 71.721]
  MoveL 2816 to (19.55, -73.22, -2.22) mm, rotated rx 180 ry 0 rz 90 deg; joints [71.682, -16.942, 81.56, 0, 25.382, 71.682]
  MoveL 2817 to (20.38, -74.49, -2.62) mm, rotated rx -180 ry 0 rz 90 deg; joints [71.651, -16.897, 81.456, 0, 25.441, 71.651]
  MoveL 2818 to (21.47, -75.55, -3.03) mm, rotated rx 180 ry 0 rz 90 deg; joints [71.629, -16.847, 81.337, 0, 25.509, 71.629]
  MoveL 2819 to (22.77, -76.34, -3.44) mm, rotated rx 180 ry 0 rz 90 deg; joints [71.618, -16.795, 81.21, 0, 25.584, 71.618]
  MoveL 2820 to (24.21, -76.82, -3.84) mm, rotated rx -180 ry 0 rz 90 deg; joints [71.618, -16.741, 81.08, 0, 25.661, 71.618]
  MoveL 2821 to (25.72, -76.95, -4.25) mm, rotated rx 180 ry 0 rz 90 deg; joints [71.629, -16.689, 80.953, 0, 25.736, 71.629]
  MoveL 2822 to (53.11, -76.67, -4.25) mm, rotated rx 180 ry 0 rz 90 deg; joints [71.916, -16.111, 78.939, 0, 27.172, 71.916]
  MoveL 2823 to (53.81, -76.63, -4.25) mm, rotated rx -180 ry 0 rz 90 deg; joints [71.924, -16.096, 78.888, 0, 27.208, 71.924]
  MoveC 2824 to (55.83, -75.42, -4.25) mm, rotated rx 180 ry 0 rz 90 deg; joints [71.982, -16.061, 78.767, 0, 27.294, 71.982] to (57.09, -73.44, -4.25) mm, rotated rx 180 ry 0 rz 90 deg; joints [72.055, -16.047, 78.72, 0, 27.327, 72.055]
  MoveC 2825 to (57.65, -71.07, -4.25) mm, rotated rx 180 ry 0 rz 90 deg; joints [72.133, -16.052, 78.736, 0, 27.316, 72.133] to (57.11, -68.7, -4.25) mm, rotated rx 180 ry 0 rz 90 deg; joints [72.201, -16.08, 78.834, 0, 27.247, 72.201]
  MoveL 2826 to (56.81, -68.32, -4.25) mm, rotated rx -180 ry 0 rz 90 deg; joints [72.209, -16.09, 78.865, 0, 27.224, 72.209]
  MoveL 2827 to (27.34, -34.24, -4.25) mm, rotated rx 180 ry 0 rz 90 deg; joints [72.982, -16.933, 81.827, 0, 25.106, 72.982]
  MoveL 2828 to (12.79, -22.61, -4.25) mm, rotated rx 180 ry 0 rz 90 deg; joints [73.211, -17.288, 83.133, 0, 24.156, 73.211]
  MoveL 2829 to (11.86, -21.94, -4.25) mm, rotated rx 180 ry 0 rz 90 deg; joints [73.223, -17.31, 83.214, 0, 24.096, 73.223]
  MoveC 2830 to (9.06, -20.95, -4.25) mm, rotated rx 180 ry 0 rz 90 deg; joints [73.228, -17.37, 83.436, 0, 23.933, 73.228] to (6.16, -21.62, -4.25) mm, rotated rx 180 ry 0 rz 90 deg; joints [73.179, -17.421, 83.629, 0, 23.792, 73.179]
  MoveC 2831 to (4.72, -22.92, -4.25) mm, rotated rx 180 ry 0 rz 90 deg; joints [73.123, -17.441, 83.703, 0, 23.738, 73.123] to (3.88, -24.67, -4.25) mm, rotated rx 180 ry 0 rz 90 deg; joints [73.059, -17.447, 83.725, 0, 23.721, 73.059]
  MoveL 2832 to (-8.38, -70.88, -4.25) mm, rotated rx 180 ry 0 rz 90 deg; joints [71.463, -17.399, 83.546, 0, 23.853, 71.463]
  MoveC 2833 to (-7.85, -74.68, -4.25) mm, rotated rx 180 ry 0 rz 90 deg; joints [71.348, -17.365, 83.418, 0, 23.947, 71.348] to (-4.76, -76.97, -4.25) mm, rotated rx -180 ry 0 rz 90 deg; joints [71.309, -17.292, 83.144, 0, 24.147, 71.309]
  MoveC 2834 to (-3.57, -77.18, -4.25) mm, rotated rx -180 ry 0 rz 90 deg; joints [71.315, -17.268, 83.055, 0, 24.212, 71.315] to (-2.37, -77.23, -4.25) mm, rotated rx 180 ry 0 rz 90 deg; joints [71.326, -17.244, 82.968, 0, 24.276, 71.326]
  MoveL 2835 to (25.72, -76.95, -4.25) mm, rotated rx 180 ry 0 rz 90 deg; joints [71.629, -16.689, 80.953, 0, 25.736, 71.629]
  MoveL 2836 to (25.64, -69.4, -4.25) mm, rotated rx 180 ry 0 rz 90 deg; joints [71.863, -16.742, 81.14, 0, 25.601, 71.863]
  MoveL 2837 to (25.64, -69.4, -1.25) mm, rotated rx 180 ry 0 rz 90 deg; joints [71.863, -16.893, 81.242, 0, 25.651, 71.863]
  Establecer velocidad (1000.0 mm/s)
  MoveL 2838 to (25.64, -69.4, 10) mm, rotated rx 180 ry 0 rz 90 deg; joints [71.863, -17.46, 81.618, 0, 25.843, 71.863]
  Establecer velocidad (66.7 mm/s)
  MoveL 2839 to (-32.42, -52.26, 10) mm, rotated rx 180 ry 0 rz 90 deg; joints [71.803, -18.679, 86.136, 0, 22.543, 71.803]
  MoveL 2840 to (-32.42, -52.26, -1) mm, rotated rx -180 ry 0 rz 90 deg; joints [71.803, -18.115, 85.77, 0, 22.344, 71.803]
  MoveL 2841 to (-31.01, -52.82, -1.41) mm, rotated rx -180 ry 0 rz 90 deg; joints [71.8, -18.066, 85.646, 0, 22.419, 71.8]
  MoveL 2842 to (-29.5, -53.02, -1.81) mm, rotated rx 180 ry 0 rz 90 deg; joints [71.809, -18.017, 85.524, 0, 22.493, 71.809]
  MoveL 2843 to (-27.99, -52.89, -2.22) mm, rotated rx -180 ry 0 rz 90 deg; joints [71.829, -17.97, 85.408, 0, 22.562, 71.829]
  MoveL 2844 to (-26.54, -52.42, -2.62) mm, rotated rx -180 ry 0 rz 90 deg; joints [71.86, -17.926, 85.304, 0, 22.622, 71.86]
  MoveL 2845 to (-25.24, -51.65, -3.03) mm, rotated rx 180 ry 0 rz 90 deg; joints [71.898, -17.887, 85.217, 0, 22.67, 71.898]
  MoveL 2846 to (-24.13, -50.6, -3.44) mm, rotated rx 180 ry 0 rz 90 deg; joints [71.944, -17.852, 85.15, 0, 22.702, 71.944]
  MoveL 2847 to (-23.29, -49.34, -3.84) mm, rotated rx -180 ry 0 rz 90 deg; joints [71.993, -17.824, 85.106, 0, 22.717, 71.993]
  MoveL 2848 to (-22.77, -47.91, -4.25) mm, rotated rx -180 ry 0 rz 90 deg; joints [72.044, -17.802, 85.089, 0, 22.713, 72.044]
  MoveL 2849 to (-16.45, -23.64, -4.25) mm, rotated rx -180 ry 0 rz 90 deg; joints [72.892, -17.826, 85.183, 0, 22.643, 72.892]
  MoveC 2850 to (-16.17, -21.53, -4.25) mm, rotated rx -180 ry 0 rz 90 deg; joints [72.963, -17.833, 85.209, 0, 22.624, 72.963] to (-16.41, -19.43, -4.25) mm, rotated rx -180 ry 0 rz 90 deg; joints [73.028, -17.849, 85.271, 0, 22.578, 73.028]
  MoveC 2851 to (-18.2, -16.69, -4.25) mm, rotated rx -180 ry 0 rz 90 deg; joints [73.1, -17.895, 85.454, 0, 22.441, 73.1] to (-21.24, -15.5, -4.25) mm, rotated rx 180 ry 0 rz 90 deg; joints [73.108, -17.955, 85.692, 0, 22.264, 73.108]
  MoveC 2852 to (-22.59, -15.51, -4.25) mm, rotated rx -180 ry 0 rz 90 deg; joints [73.095, -17.979, 85.785, 0, 22.194, 73.095] to (-23.92, -15.7, -4.25) mm, rotated rx -180 ry 0 rz 90 deg; joints [73.075, -18.001, 85.874, 0, 22.127, 73.075]
  MoveL 2853 to (-72.88, -26.13, -4.25) mm, rotated rx -180 ry 0 rz 90 deg; joints [72.229, -18.751, 88.994, 0, 19.757, 72.229]
  MoveC 2854 to (-76.52, -28.36, -4.25) mm, rotated rx 180 ry 0 rz 90 deg; joints [72.115, -18.796, 89.189, 0, 19.607, 72.115] to (-77.94, -32.38, -4.25) mm, rotated rx 180 ry 0 rz 90 deg; joints [71.966, -18.798, 89.198, 0, 19.6, 71.966]
  MoveL 2855 to (-77.94, -71.02, -4.25) mm, rotated rx 180 ry 0 rz 90 deg; joints [70.69, -18.596, 88.325, 0, 20.271, 70.69]
  MoveC 2856 to (-76.23, -75.31, -4.25) mm, rotated rx 180 ry 0 rz 90 deg; joints [70.569, -18.546, 88.109, 0, 20.436, 70.569] to (-72.02, -77.24, -4.25) mm, rotated rx -180 ry 0 rz 90 deg; joints [70.554, -18.468, 87.782, 0, 20.686, 70.554]
  MoveL 2857 to (-70.6, -77.31, -4.25) mm, rotated rx 180 ry 0 rz 90 deg; joints [70.569, -18.445, 87.684, 0, 20.761, 70.569]
  MoveL 2858 to (-35.31, -77.03, -4.25) mm, rotated rx -180 ry 0 rz 90 deg; joints [70.975, -17.852, 85.284, 0, 22.568, 70.975]
  MoveC 2859 to (-31.38, -75.66, -4.25) mm, rotated rx -180 ry 0 rz 90 deg; joints [71.062, -17.791, 85.044, 0, 22.746, 71.062] to (-29.1, -72.19, -4.25) mm, rotated rx 180 ry 0 rz 90 deg; joints [71.198, -17.771, 84.968, 0, 22.803, 71.198]
  MoveL 2860 to (-22.77, -47.91, -4.25) mm, rotated rx -180 ry 0 rz 90 deg; joints [72.044, -17.802, 85.089, 0, 22.713, 72.044]
  MoveL 2861 to (-30.08, -46.01, -4.25) mm, rotated rx -180 ry 0 rz 90 deg; joints [72.029, -17.942, 85.64, 0, 22.302, 72.029]
  MoveL 2862 to (-30.08, -46.01, -1.25) mm, rotated rx 180 ry 0 rz 90 deg; joints [72.029, -18.096, 85.741, 0, 22.355, 72.029]
  Establecer velocidad (1000.0 mm/s)
  MoveL 2863 to (-30.08, -46.01, 10) mm, rotated rx 180 ry 0 rz 90 deg; joints [72.029, -18.674, 86.116, 0, 22.558, 72.029]
  Establecer velocidad (66.7 mm/s)
  MoveL 2864 to (-69.71, 36.15, 10) mm, rotated rx 180 ry 0 rz 90 deg; joints [74.354, -19.732, 90.51, 0, 19.222, 74.354]
  MoveL 2865 to (-69.71, 36.15, -1) mm, rotated rx -180 ry 0 rz 90 deg; joints [74.354, -19.156, 90.143, 0, 19.012, 74.354]
  MoveL 2866 to (-71.21, 36.33, -1.41) mm, rotated rx -180 ry 0 rz 90 deg; joints [74.346, -19.158, 90.234, 0, 18.924, 74.346]
  MoveL 2867 to (-72.72, 36.15, -1.81) mm, rotated rx 180 ry 0 rz 90 deg; joints [74.326, -19.158, 90.318, 0, 18.84, 74.326]
  MoveL 2868 to (-74.15, 35.64, -2.22) mm, rotated rx 180 ry 0 rz 90 deg; joints [74.294, -19.156, 90.39, 0, 18.765, 74.294]
  MoveL 2869 to (-75.43, 34.82, -2.62) mm, rotated rx 180 ry 0 rz 90 deg; joints [74.254, -19.15, 90.447, 0, 18.703, 74.254]
  MoveL 2870 to (-76.5, 33.74, -3.03) mm, rotated rx 180 ry 0 rz 90 deg; joints [74.207, -19.14, 90.484, 0, 18.655, 74.207]
  MoveL 2871 to (-77.3, 32.46, -3.44) mm, rotated rx -180 ry 0 rz 90 deg; joints [74.156, -19.125, 90.5, 0, 18.625, 74.156]
  MoveL 2872 to (-77.81, 31.02, -3.84) mm, rotated rx 180 ry 0 rz 90 deg; joints [74.102, -19.105, 90.492, 0, 18.612, 74.102]
  MoveL 2873 to (-77.94, 29.51, -4.25) mm, rotated rx -180 ry 0 rz 90 deg; joints [74.049, -19.079, 90.459, 0, 18.62, 74.049]
  MoveL 2874 to (-77.94, 1.42, -4.25) mm, rotated rx -180 ry 0 rz 90 deg; joints [73.098, -18.958, 89.907, 0, 19.05, 73.098]
  MoveL 2875 to (-77.94, 0.3, -4.25) mm, rotated rx -180 ry 0 rz 90 deg; joints [73.06, -18.952, 89.884, 0, 19.068, 73.06]
  MoveC 2876 to (-76.5, -3.59, -4.25) mm, rotated rx 180 ry 0 rz 90 deg; joints [72.944, -18.913, 89.708, 0, 19.205, 72.944] to (-72.89, -5.63, -4.25) mm, rotated rx 180 ry 0 rz 90 deg; joints [72.913, -18.85, 89.426, 0, 19.424, 72.913]
  MoveC 2877 to (-71.27, -5.73, -4.25) mm, rotated rx 180 ry 0 rz 90 deg; joints [72.926, -18.824, 89.315, 0, 19.51, 72.926] to (-69.65, -5.51, -4.25) mm, rotated rx -180 ry 0 rz 90 deg; joints [72.95, -18.801, 89.211, 0, 19.59, 72.95]
  MoveL 2878 to (-20.08, 5.89, -4.25) mm, rotated rx 180 ry 0 rz 90 deg; joints [73.817, -18.046, 86.053, 0, 21.993, 73.817]
  MoveC 2879 to (-17.67, 7.01, -4.25) mm, rotated rx -180 ry 0 rz 90 deg; joints [73.877, -18.01, 85.908, 0, 22.102, 73.877] to (-15.93, 9, -4.25) mm, rotated rx 180 ry 0 rz 90 deg; joints [73.958, -17.989, 85.826, 0, 22.163, 73.958]
  MoveC 2880 to (-15.28, 11.37, -4.25) mm, rotated rx 180 ry 0 rz 90 deg; joints [74.042, -17.99, 85.829, 0, 22.161, 74.042] to (-15.55, 13.82, -4.25) mm, rotated rx -180 ry 0 rz 90 deg; joints [74.119, -18.007, 85.897, 0, 22.11, 74.119]
  MoveL 2881 to (-15.82, 14.69, -4.25) mm, rotated rx 180 ry 0 rz 90 deg; joints [74.145, -18.016, 85.933, 0, 22.083, 74.145]
  MoveL 2882 to (-22.49, 33.31, -4.25) mm, rotated rx 180 ry 0 rz 90 deg; joints [74.697, -18.221, 86.759, 0, 21.462, 74.697]
  MoveC 2883 to (-23.54, 35.19, -4.25) mm, rotated rx 180 ry 0 rz 90 deg; joints [74.75, -18.248, 86.868, 0, 21.38, 74.75] to (-25.13, 36.63, -4.25) mm, rotated rx -180 ry 0 rz 90 deg; joints [74.783, -18.281, 87.006, 0, 21.276, 74.783]
  MoveL 2884 to (-66.81, 63.38, -4.25) mm, rotated rx 180 ry 0 rz 90 deg; joints [75.309, -19.052, 90.335, 0, 18.717, 75.309]
  MoveL 2885 to (-67.76, 63.95, -4.25) mm, rotated rx -180 ry 0 rz 90 deg; joints [75.32, -19.068, 90.409, 0, 18.659, 75.32]
  MoveC 2886 to (-69.91, 64.94, -4.25) mm, rotated rx 180 ry 0 rz 90 deg; joints [75.334, -19.103, 90.57, 0, 18.533, 75.334] to (-72.25, 65.35, -4.25) mm, rotated rx 180 ry 0 rz 90 deg; joints [75.328, -19.139, 90.733, 0, 18.405, 75.328]
  MoveC 2887 to (-75.22, 64.57, -4.25) mm, rotated rx -180 ry 0 rz 90 deg; joints [75.274, -19.178, 90.919, 0, 18.26, 75.274] to (-77.23, 62.24, -4.25) mm, rotated rx 180 ry 0 rz 90 deg; joints [75.175, -19.198, 91.011, 0, 18.187, 75.175]
  MoveC 2888 to (-77.76, 60.52, -4.25) mm, rotated rx -180 ry 0 rz 90 deg; joints [75.111, -19.199, 91.016, 0, 18.183, 75.111] to (-77.94, 58.72, -4.25) mm, rotated rx 180 ry 0 rz 90 deg; joints [75.048, -19.195, 90.997, 0, 18.198, 75.048]
  MoveL 2889 to (-77.94, 29.51, -4.25) mm, rotated rx -180 ry 0 rz 90 deg; joints [74.049, -19.079, 90.459, 0, 18.62, 74.049]
  MoveL 2890 to (-70.39, 29.51, -4.25) mm, rotated rx -180 ry 0 rz 90 deg; joints [74.122, -18.968, 89.955, 0, 19.013, 74.122]
  MoveL 2891 to (-70.39, 29.51, -1.25) mm, rotated rx -180 ry 0 rz 90 deg; joints [74.122, -19.125, 90.056, 0, 19.07, 74.122]
  Establecer velocidad (1000.0 mm/s)
  MoveL 2892 to (-70.39, 29.51, 10) mm, rotated rx 180 ry 0 rz 90 deg; joints [74.122, -19.714, 90.43, 0, 19.284, 74.122]
  Establecer velocidad (66.7 mm/s)
  MoveL 2893 to (-69.42, 36.15, 10) mm, rotated rx -180 ry 0 rz 90 deg; joints [74.357, -19.728, 90.491, 0, 19.237, 74.357]
  MoveL 2894 to (-69.42, 36.15, -1.25) mm, rotated rx -180 ry 0 rz 90 deg; joints [74.357, -19.139, 90.116, 0, 19.022, 74.357]
  MoveL 2895 to (-70.93, 36.33, -1.66) mm, rotated rx 180 ry 0 rz 90 deg; joints [74.349, -19.141, 90.207, 0, 18.934, 74.349]
  MoveL 2896 to (-72.44, 36.15, -2.06) mm, rotated rx 180 ry 0 rz 90 deg; joints [74.328, -19.141, 90.291, 0, 18.85, 74.328]
  MoveL 2897 to (-73.87, 35.64, -2.47) mm, rotated rx 180 ry 0 rz 90 deg; joints [74.297, -19.138, 90.363, 0, 18.775, 74.297]
  MoveL 2898 to (-75.15, 34.82, -2.88) mm, rotated rx -180 ry 0 rz 90 deg; joints [74.257, -19.132, 90.42, 0, 18.713, 74.257]
  MoveL 2899 to (-76.22, 33.74, -3.28) mm, rotated rx 180 ry 0 rz 90 deg; joints [74.21, -19.122, 90.457, 0, 18.665, 74.21]
  MoveL 2900 to (-77.03, 32.46, -3.69) mm, rotated rx -180 ry 0 rz 90 deg; joints [74.158, -19.107, 90.473, 0, 18.635, 74.158]
  MoveL 2901 to (-77.52, 31.02, -4.09) mm, rotated rx -180 ry 0 rz 90 deg; joints [74.105, -19.087, 90.465, 0, 18.622, 74.105]
  MoveL 2902 to (-77.66, 29.51, -4.5) mm, rotated rx 180 ry 0 rz 90 deg; joints [74.052, -19.062, 90.432, 0, 18.63, 74.052]
  MoveL 2903 to (-77.66, 1.42, -4.5) mm, rotated rx 180 ry 0 rz 90 deg; joints [73.101, -18.94, 89.88, 0, 19.06, 73.101]
  MoveL 2904 to (-77.66, 0.32, -4.5) mm, rotated rx -180 ry 0 rz 90 deg; joints [73.064, -18.935, 89.857, 0, 19.078, 73.064]
  MoveC 2905 to (-76.19, -3.49, -4.5) mm, rotated rx -180 ry 0 rz 90 deg; joints [72.951, -18.896, 89.682, 0, 19.214, 72.951] to (-72.57, -5.39, -4.5) mm, rotated rx 180 ry 0 rz 90 deg; joints [72.924, -18.833, 89.401, 0, 19.432, 72.924]
  MoveC 2906 to (-71.1, -5.43, -4.5) mm, rotated rx 180 ry 0 rz 90 deg; joints [72.938, -18.81, 89.301, 0, 19.509, 72.938] to (-69.65, -5.21, -4.5) mm, rotated rx 180 ry 0 rz 90 deg; joints [72.96, -18.789, 89.209, 0, 19.58, 72.96]
  MoveL 2907 to (-20.37, 6.13, -4.5) mm, rotated rx 180 ry 0 rz 90 deg; joints [73.822, -18.04, 86.07, 0, 21.969, 73.822]
  MoveL 2908 to (-20.27, 6.16, -4.5) mm, rotated rx -180 ry 0 rz 90 deg; joints [73.824, -18.038, 86.064, 0, 21.974, 73.824]
  MoveL 2909 to (-19.43, 6.4, -4.5) mm, rotated rx 180 ry 0 rz 90 deg; joints [73.84, -18.024, 86.01, 0, 22.015, 73.84]
  MoveC 2910 to (-16.34, 8.89, -4.5) mm, rotated rx -180 ry 0 rz 90 deg; joints [73.951, -17.983, 85.844, 0, 22.139, 73.951] to (-15.63, 12.79, -4.5) mm, rotated rx -180 ry 0 rz 90 deg; joints [74.085, -17.99, 85.873, 0, 22.117, 74.085]
  MoveL 2911 to (-15.86, 13.92, -4.5) mm, rotated rx -180 ry 0 rz 90 deg; joints [74.12, -18, 85.912, 0, 22.088, 74.12]
  MoveC 2912 to (-15.9, 14.07, -4.5) mm, rotated rx -180 ry 0 rz 90 deg; joints [74.124, -18.001, 85.918, 0, 22.084, 74.124] to (-15.95, 14.22, -4.5) mm, rotated rx -180 ry 0 rz 90 deg; joints [74.129, -18.003, 85.924, 0, 22.079, 74.129]
  MoveL 2913 to (-22.72, 33.13, -4.5) mm, rotated rx 180 ry 0 rz 90 deg; joints [74.689, -18.211, 86.763, 0, 21.448, 74.689]
  MoveC 2914 to (-23.75, 34.99, -4.5) mm, rotated rx 180 ry 0 rz 90 deg; joints [74.741, -18.237, 86.87, 0, 21.367, 74.741] to (-25.32, 36.41, -4.5) mm, rotated rx 180 ry 0 rz 90 deg; joints [74.774, -18.27, 87.006, 0, 21.265, 74.774]
  MoveL 2915 to (-28.38, 38.38, -4.5) mm, rotated rx 180 ry 0 rz 90 deg; joints [74.812, -18.331, 87.255, 0, 21.076, 74.812]
  MoveL 2916 to (-67.76, 63.63, -4.5) mm, rotated rx 180 ry 0 rz 90 deg; joints [75.309, -19.054, 90.394, 0, 18.659, 75.309]
  MoveC 2917 to (-69.9, 64.63, -4.5) mm, rotated rx -180 ry 0 rz 90 deg; joints [75.324, -19.089, 90.555, 0, 18.533, 75.324] to (-72.22, 65.06, -4.5) mm, rotated rx 180 ry 0 rz 90 deg; joints [75.318, -19.124, 90.718, 0, 18.406, 75.318]
  MoveC 2918 to (-75.11, 64.3, -4.5) mm, rotated rx -180 ry 0 rz 90 deg; joints [75.266, -19.162, 90.898, 0, 18.265, 75.266] to (-77.02, 62, -4.5) mm, rotated rx 180 ry 0 rz 90 deg; joints [75.169, -19.181, 90.984, 0, 18.197, 75.169]
  MoveC 2919 to (-77.5, 60.36, -4.5) mm, rotated rx -180 ry 0 rz 90 deg; joints [75.108, -19.182, 90.988, 0, 18.194, 75.108] to (-77.66, 58.66, -4.5) mm, rotated rx -180 ry 0 rz 90 deg; joints [75.048, -19.178, 90.968, 0, 18.209, 75.048]
  MoveL 2920 to (-77.66, 29.51, -4.5) mm, rotated rx 180 ry 0 rz 90 deg; joints [74.052, -19.062, 90.432, 0, 18.63, 74.052]
  MoveL 2921 to (-70.11, 29.51, -4.5) mm, rotated rx -180 ry 0 rz 90 deg; joints [74.125, -18.951, 89.927, 0, 19.023, 74.125]
  MoveL 2922 to (-70.11, 29.51, -1.5) mm, rotated rx 180 ry 0 rz 90 deg; joints [74.125, -19.108, 90.028, 0, 19.079, 74.125]
  Establecer velocidad (1000.0 mm/s)
  MoveL 2923 to (-70.11, 29.51, 10) mm, rotated rx 180 ry 0 rz 90 deg; joints [74.125, -19.71, 90.412, 0, 19.298, 74.125]
  Establecer velocidad (66.7 mm/s)
  MoveL 2924 to (-40.16, -27.87, 10) mm, rotated rx -180 ry 0 rz 90 deg; joints [72.514, -18.951, 87.212, 0, 21.739, 72.514]
  MoveL 2925 to (-40.16, -27.87, -1.25) mm, rotated rx -180 ry 0 rz 90 deg; joints [72.514, -18.37, 86.837, 0, 21.533, 72.514]
  MoveL 2926 to (-40.29, -26.36, -1.66) mm, rotated rx 180 ry 0 rz 90 deg; joints [72.562, -18.36, 86.866, 0, 21.494, 72.562]
  MoveL 2927 to (-40.78, -24.92, -2.06) mm, rotated rx 180 ry 0 rz 90 deg; joints [72.604, -18.354, 86.917, 0, 21.438, 72.604]
  MoveL 2928 to (-41.58, -23.62, -2.47) mm, rotated rx 180 ry 0 rz 90 deg; joints [72.638, -18.354, 86.986, 0, 21.368, 72.638]
  MoveL 2929 to (-42.65, -22.54, -2.88) mm, rotated rx -180 ry 0 rz 90 deg; joints [72.663, -18.356, 87.068, 0, 21.288, 72.663]
  MoveL 2930 to (-43.93, -21.72, -3.28) mm, rotated rx 180 ry 0 rz 90 deg; joints [72.677, -18.361, 87.16, 0, 21.201, 72.677]
  MoveL 2931 to (-45.35, -21.2, -3.69) mm, rotated rx -180 ry 0 rz 90 deg; joints [72.679, -18.366, 87.255, 0, 21.111, 72.679]
  MoveL 2932 to (-46.86, -21.01, -4.09) mm, rotated rx -180 ry 0 rz 90 deg; joints [72.67, -18.371, 87.348, 0, 21.023, 72.67]
  MoveL 2933 to (-48.37, -21.19, -4.5) mm, rotated rx -180 ry 0 rz 90 deg; joints [72.649, -18.374, 87.434, 0, 20.94, 72.649]
  MoveL 2934 to (-72.79, -26.39, -4.5) mm, rotated rx -180 ry 0 rz 90 deg; joints [72.221, -18.736, 88.974, 0, 19.762, 72.221]
  MoveC 2935 to (-76.29, -28.53, -4.5) mm, rotated rx 180 ry 0 rz 90 deg; joints [72.112, -18.779, 89.162, 0, 19.617, 72.112] to (-77.66, -32.41, -4.5) mm, rotated rx -180 ry 0 rz 90 deg; joints [71.968, -18.78, 89.17, 0, 19.611, 71.968]
  MoveL 2936 to (-77.66, -70.81, -4.5) mm, rotated rx -180 ry 0 rz 90 deg; joints [70.7, -18.58, 88.303, 0, 20.277, 70.7]
  MoveC 2937 to (-77.4, -72.67, -4.5) mm, rotated rx -180 ry 0 rz 90 deg; joints [70.642, -18.566, 88.241, 0, 20.324, 70.642] to (-76.63, -74.39, -4.5) mm, rotated rx 180 ry 0 rz 90 deg; joints [70.594, -18.544, 88.149, 0, 20.395, 70.594]
  MoveC 2938 to (-74.4, -76.31, -4.5) mm, rotated rx 180 ry 0 rz 90 deg; joints [70.557, -18.498, 87.955, 0, 20.543, 70.557] to (-71.55, -77.02, -4.5) mm, rotated rx -180 ry 0 rz 90 deg; joints [70.567, -18.449, 87.746, 0, 20.702, 70.567]
  MoveL 2939 to (-70.6, -77.03, -4.5) mm, rotated rx -180 ry 0 rz 90 deg; joints [70.578, -18.433, 87.682, 0, 20.751, 70.578]
  MoveL 2940 to (-42.17, -76.81, -4.5) mm, rotated rx 180 ry 0 rz 90 deg; joints [70.906, -17.96, 85.754, 0, 22.206, 70.906]
  MoveL 2941 to (-35.31, -76.75, -4.5) mm, rotated rx 180 ry 0 rz 90 deg; joints [70.984, -17.841, 85.282, 0, 22.559, 70.984]
  MoveC 2942 to (-31.56, -75.44, -4.5) mm, rotated rx 180 ry 0 rz 90 deg; joints [71.067, -17.782, 85.053, 0, 22.729, 71.067] to (-29.38, -72.12, -4.5) mm, rotated rx -180 ry 0 rz 90 deg; joints [71.197, -17.764, 84.981, 0, 22.783, 71.197]
  MoveL 2943 to (-16.81, -23.95, -4.5) mm, rotated rx -180 ry 0 rz 90 deg; joints [72.878, -17.818, 85.193, 0, 22.625, 72.878]
  MoveC 2944 to (-16.5, -22.04, -4.5) mm, rotated rx 180 ry 0 rz 90 deg; joints [72.943, -17.823, 85.213, 0, 22.61, 72.943] to (-16.58, -20.1, -4.5) mm, rotated rx 180 ry 0 rz 90 deg; joints [73.005, -17.835, 85.26, 0, 22.575, 73.005]
  MoveC 2945 to (-18.17, -17.09, -4.5) mm, rotated rx 180 ry 0 rz 90 deg; joints [73.087, -17.88, 85.435, 0, 22.444, 73.087] to (-21.31, -15.78, -4.5) mm, rotated rx 180 ry 0 rz 90 deg; joints [73.098, -17.942, 85.682, 0, 22.26, 73.098]
  MoveC 2946 to (-22.64, -15.8, -4.5) mm, rotated rx 180 ry 0 rz 90 deg; joints [73.084, -17.965, 85.774, 0, 22.191, 73.084] to (-23.95, -15.99, -4.5) mm, rotated rx 180 ry 0 rz 90 deg; joints [73.065, -17.987, 85.861, 0, 22.126, 73.065]
  MoveL 2947 to (-48.37, -21.19, -4.5) mm, rotated rx -180 ry 0 rz 90 deg; joints [72.649, -18.374, 87.434, 0, 20.94, 72.649]
  MoveL 2948 to (-46.8, -28.57, -4.5) mm, rotated rx 180 ry 0 rz 90 deg; joints [72.422, -18.31, 87.168, 0, 21.142, 72.422]
  MoveL 2949 to (-46.8, -28.57, -1.5) mm, rotated rx -180 ry 0 rz 90 deg; joints [72.422, -18.465, 87.269, 0, 21.196, 72.422]
  Establecer velocidad (1000.0 mm/s)
  MoveL 2950 to (-46.8, -28.57, 10) mm, rotated rx 180 ry 0 rz 90 deg; joints [72.422, -19.059, 87.651, 0, 21.408, 72.422]
  Establecer velocidad (66.7 mm/s)
  MoveL 2951 to (18.86, -68.5, 10) mm, rotated rx 180 ry 0 rz 90 deg; joints [71.822, -17.605, 82.131, 0, 25.474, 71.822]
  MoveL 2952 to (18.86, -68.5, -1.25) mm, rotated rx -180 ry 0 rz 90 deg; joints [71.822, -17.037, 81.755, 0, 25.281, 71.822]
  MoveL 2953 to (18.69, -70, -1.66) mm, rotated rx 180 ry 0 rz 90 deg; joints [71.773, -17.009, 81.718, 0, 25.291, 71.773]
  MoveL 2954 to (18.89, -71.51, -2.06) mm, rotated rx 180 ry 0 rz 90 deg; joints [71.728, -16.975, 81.654, 0, 25.321, 71.728]
  MoveL 2955 to (19.42, -72.94, -2.47) mm, rotated rx -180 ry 0 rz 90 deg; joints [71.689, -16.934, 81.568, 0, 25.366, 71.689]
  MoveL 2956 to (20.25, -74.21, -2.88) mm, rotated rx -180 ry 0 rz 90 deg; joints [71.658, -16.888, 81.464, 0, 25.425, 71.658]
  MoveL 2957 to (21.34, -75.27, -3.28) mm, rotated rx 180 ry 0 rz 90 deg; joints [71.636, -16.839, 81.345, 0, 25.493, 71.636]
  MoveL 2958 to (22.63, -76.06, -3.69) mm, rotated rx -180 ry 0 rz 90 deg; joints [71.625, -16.786, 81.218, 0, 25.568, 71.625]
  MoveL 2959 to (24.07, -76.54, -4.09) mm, rotated rx -180 ry 0 rz 90 deg; joints [71.625, -16.733, 81.088, 0, 25.645, 71.625]
  MoveL 2960 to (25.59, -76.67, -4.5) mm, rotated rx 180 ry 0 rz 90 deg; joints [71.637, -16.681, 80.961, 0, 25.72, 71.637]
  MoveL 2961 to (53.07, -76.38, -4.5) mm, rotated rx 180 ry 0 rz 90 deg; joints [71.925, -16.102, 78.941, 0, 27.161, 71.925]
  MoveL 2962 to (53.54, -76.35, -4.5) mm, rotated rx 180 ry 0 rz 90 deg; joints [71.93, -16.092, 78.906, 0, 27.185, 71.93]
  MoveC 2963 to (54.62, -75.76, -4.5) mm, rotated rx 180 ry 0 rz 90 deg; joints [71.959, -16.072, 78.84, 0, 27.232, 71.959] to (55.51, -74.91, -4.5) mm, rotated rx 180 ry 0 rz 90 deg; joints [71.994, -16.059, 78.794, 0, 27.264, 71.994]
  MoveL 2964 to (55.74, -74.62, -4.5) mm, rotated rx -180 ry 0 rz 90 deg; joints [72.005, -16.056, 78.784, 0, 27.272, 72.005]
  MoveC 2965 to (57, -71.79, -4.5) mm, rotated rx -180 ry 0 rz 90 deg; joints [72.105, -16.048, 78.758, 0, 27.29, 72.105] to (56.73, -68.7, -4.5) mm, rotated rx 180 ry 0 rz 90 deg; joints [72.197, -16.076, 78.853, 0, 27.223, 72.197]
  MoveL 2966 to (56.57, -68.48, -4.5) mm, rotated rx 180 ry 0 rz 90 deg; joints [72.202, -16.081, 78.871, 0, 27.21, 72.202]
  MoveL 2967 to (27.96, -35.37, -4.5) mm, rotated rx -180 ry 0 rz 90 deg; joints [72.953, -16.901, 81.749, 0, 25.152, 72.953]
  MoveL 2968 to (27.13, -34.46, -4.5) mm, rotated rx 180 ry 0 rz 90 deg; joints [72.973, -16.923, 81.829, 0, 25.094, 72.973]
  MoveL 2969 to (12.79, -22.98, -4.5) mm, rotated rx 180 ry 0 rz 90 deg; joints [73.199, -17.274, 83.116, 0, 24.157, 73.199]
  MoveC 2970 to (12, -22.4, -4.5) mm, rotated rx -180 ry 0 rz 90 deg; joints [73.21, -17.292, 83.186, 0, 24.107, 73.21] to (11.16, -21.89, -4.5) mm, rotated rx 180 ry 0 rz 90 deg; joints [73.218, -17.311, 83.257, 0, 24.054, 73.218]
  MoveC 2971 to (7.9, -21.37, -4.5) mm, rotated rx -180 ry 0 rz 90 deg; joints [73.203, -17.376, 83.501, 0, 23.875, 73.203] to (5.04, -23.01, -4.5) mm, rotated rx -180 ry 0 rz 90 deg; joints [73.123, -17.421, 83.67, 0, 23.752, 73.123]
  MoveC 2972 to (4.45, -24.02, -4.5) mm, rotated rx 180 ry 0 rz 90 deg; joints [73.085, -17.427, 83.69, 0, 23.737, 73.085] to (4.07, -25.11, -4.5) mm, rotated rx 180 ry 0 rz 90 deg; joints [73.046, -17.428, 83.694, 0, 23.734, 73.046]
  MoveL 2973 to (-8.08, -70.88, -4.5) mm, rotated rx 180 ry 0 rz 90 deg; joints [71.466, -17.38, 83.516, 0, 23.864, 71.466]
  MoveC 2974 to (-7.61, -74.46, -4.5) mm, rotated rx 180 ry 0 rz 90 deg; joints [71.358, -17.349, 83.398, 0, 23.951, 71.358] to (-4.75, -76.67, -4.5) mm, rotated rx 180 ry 0 rz 90 deg; joints [71.318, -17.281, 83.143, 0, 24.138, 71.318]
  MoveC 2975 to (-3.57, -76.9, -4.5) mm, rotated rx 180 ry 0 rz 90 deg; joints [71.323, -17.257, 83.053, 0, 24.203, 71.323] to (-2.37, -76.96, -4.5) mm, rotated rx 180 ry 0 rz 90 deg; joints [71.334, -17.233, 82.966, 0, 24.267, 71.334]
  MoveL 2976 to (25.59, -76.67, -4.5) mm, rotated rx 180 ry 0 rz 90 deg; joints [71.637, -16.681, 80.961, 0, 25.72, 71.637]
  MoveL 2977 to (25.51, -69.12, -4.5) mm, rotated rx 180 ry 0 rz 90 deg; joints [71.871, -16.733, 81.148, 0, 25.585, 71.871]
  MoveL 2978 to (25.51, -69.12, -1.5) mm, rotated rx 180 ry 0 rz 90 deg; joints [71.871, -16.885, 81.25, 0, 25.635, 71.871]
  Establecer velocidad (1000.0 mm/s)
  MoveL 2979 to (25.51, -69.12, 10) mm, rotated rx 180 ry 0 rz 90 deg; joints [71.871, -17.465, 81.635, 0, 25.831, 71.871]
  Establecer velocidad (66.7 mm/s)
  MoveL 2980 to (66.95, -31.01, 10) mm, rotated rx 180 ry 0 rz 90 deg; joints [73.456, -16.834, 79.449, 0, 27.385, 73.456]
  MoveL 2981 to (66.95, -31.01, -1.25) mm, rotated rx 180 ry 0 rz 90 deg; joints [73.456, -16.27, 79.071, 0, 27.199, 73.456]
  MoveL 2982 to (68.46, -31.2, -1.66) mm, rotated rx 180 ry 0 rz 90 deg; joints [73.464, -16.216, 78.94, 0, 27.276, 73.464]
  MoveL 2983 to (69.96, -31.02, -2.06) mm, rotated rx -180 ry 0 rz 90 deg; joints [73.484, -16.163, 78.816, 0, 27.347, 73.484]
  MoveL 2984 to (71.39, -30.51, -2.47) mm, rotated rx -180 ry 0 rz 90 deg; joints [73.513, -16.114, 78.706, 0, 27.409, 73.513]
  MoveL 2985 to (72.68, -29.69, -2.88) mm, rotated rx -180 ry 0 rz 90 deg; joints [73.549, -16.071, 78.613, 0, 27.458, 73.549]
  MoveL 2986 to (73.75, -28.61, -3.28) mm, rotated rx -180 ry 0 rz 90 deg; joints [73.593, -16.034, 78.543, 0, 27.491, 73.593]
  MoveL 2987 to (74.55, -27.32, -3.69) mm, rotated rx -180 ry 0 rz 90 deg; joints [73.64, -16.004, 78.496, 0, 27.507, 73.64]
  MoveL 2988 to (75.05, -25.89, -4.09) mm, rotated rx -180 ry 0 rz 90 deg; joints [73.688, -15.982, 78.476, 0, 27.505, 73.688]
  MoveL 2989 to (75.19, -24.37, -4.5) mm, rotated rx -180 ry 0 rz 90 deg; joints [73.736, -15.968, 78.486, 0, 27.482, 73.736]
  MoveL 2990 to (75.19, -5.9, -4.5) mm, rotated rx 180 ry 0 rz 90 deg; joints [74.308, -16.086, 78.886, 0, 27.199, 74.308]
  MoveC 2991 to (72.95, -3.07, -4.5) mm, rotated rx 180 ry 0 rz 90 deg; joints [74.377, -16.153, 79.115, 0, 27.037, 74.377] to (69.65, -1.61, -4.5) mm, rotated rx 180 ry 0 rz 90 deg; joints [74.394, -16.234, 79.395, 0, 26.839, 74.394]
  MoveC 2992 to (68.27, -1.59, -4.5) mm, rotated rx 180 ry 0 rz 90 deg; joints [74.382, -16.264, 79.499, 0, 26.765, 74.382] to (66.96, -1.99, -4.5) mm, rotated rx -180 ry 0 rz 90 deg; joints [74.358, -16.29, 79.589, 0, 26.701, 74.358]
  MoveL 2993 to (66.81, -2.19, -4.5) mm, rotated rx -180 ry 0 rz 90 deg; joints [74.351, -16.292, 79.596, 0, 26.696, 74.351]
  MoveL 2994 to (51.35, -23.38, -4.5) mm, rotated rx 180 ry 0 rz 90 deg; joints [73.55, -16.492, 80.295, 0, 26.197, 73.55]
  MoveC 2995 to (50.5, -26.23, -4.5) mm, rotated rx 180 ry 0 rz 90 deg; joints [73.453, -16.493, 80.296, 0, 26.197, 73.453] to (51.62, -28.98, -4.5) mm, rotated rx 180 ry 0 rz 90 deg; joints [73.377, -16.452, 80.152, 0, 26.3, 73.377]
  MoveL 2996 to (67.28, -46.69, -4.5) mm, rotated rx -180 ry 0 rz 90 deg; joints [72.975, -15.996, 78.579, 0, 27.416, 72.975]
  MoveC 2997 to (68.42, -47.14, -4.5) mm, rotated rx 180 ry 0 rz 90 deg; joints [72.972, -15.967, 78.483, 0, 27.485, 72.972] to (69.65, -47.16, -4.5) mm, rotated rx 180 ry 0 rz 90 deg; joints [72.983, -15.94, 78.389, 0, 27.55, 72.983]
  MoveC 2998 to (73, -45.75, -4.5) mm, rotated rx 180 ry 0 rz 90 deg; joints [73.058, -15.875, 78.169, 0, 27.706, 73.058] to (75.19, -42.85, -4.5) mm, rotated rx 180 ry 0 rz 90 deg; joints [73.168, -15.845, 78.069, 0, 27.776, 73.168]
  MoveL 2999 to (75.19, -24.37, -4.5) mm, rotated rx -180 ry 0 rz 90 deg; joints [73.736, -15.968, 78.486, 0, 27.482, 73.736]
  MoveL 3000 to (67.64, -24.37, -4.5) mm, rotated rx -180 ry 0 rz 90 deg; joints [73.668, -16.135, 79.056, 0, 27.079, 73.668]
  MoveL 3001 to (67.64, -24.37, -1.5) mm, rotated rx 180 ry 0 rz 90 deg; joints [73.668, -16.286, 79.158, 0, 27.128, 73.668]
  Establecer velocidad (1000.0 mm/s)
  MoveL 3002 to (67.64, -24.37, 10) mm, rotated rx -180 ry 0 rz 90 deg; joints [73.668, -16.862, 79.544, 0, 27.317, 73.668]
  Establecer velocidad (66.7 mm/s)
  MoveL 3003 to (35.63, 8.63, 10) mm, rotated rx -180 ry 0 rz 90 deg; joints [74.417, -17.739, 82.613, 0, 25.126, 74.417]
  MoveL 3004 to (35.63, 8.63, -1.25) mm, rotated rx 180 ry 0 rz 90 deg; joints [74.417, -17.17, 82.237, 0, 24.932, 74.417]
  MoveL 3005 to (36.75, 7.6, -1.66) mm, rotated rx 180 ry 0 rz 90 deg; joints [74.394, -17.121, 82.121, 0, 25, 74.394]
  MoveL 3006 to (38.08, 6.87, -2.06) mm, rotated rx 180 ry 0 rz 90 deg; joints [74.383, -17.07, 81.995, 0, 25.074, 74.383]
  MoveL 3007 to (39.54, 6.45, -2.47) mm, rotated rx 180 ry 0 rz 90 deg; joints [74.383, -17.017, 81.866, 0, 25.151, 74.383]
  MoveL 3008 to (41.06, 6.37, -2.88) mm, rotated rx 180 ry 0 rz 90 deg; joints [74.393, -16.965, 81.74, 0, 25.226, 74.393]
  MoveL 3009 to (42.56, 6.62, -3.28) mm, rotated rx 180 ry 0 rz 90 deg; joints [74.415, -16.915, 81.621, 0, 25.295, 74.415]
  MoveL 3010 to (43.96, 7.2, -3.69) mm, rotated rx -180 ry 0 rz 90 deg; joints [74.445, -16.87, 81.516, 0, 25.354, 74.445]
  MoveL 3011 to (45.2, 8.07, -4.09) mm, rotated rx -180 ry 0 rz 90 deg; joints [74.484, -16.829, 81.429, 0, 25.4, 74.484]
  MoveL 3012 to (46.2, 9.22, -4.5) mm, rotated rx 180 ry 0 rz 90 deg; joints [74.529, -16.794, 81.365, 0, 25.429, 74.529]
  MoveL 3013 to (57.76, 25.32, -4.5) mm, rotated rx -180 ry 0 rz 90 deg; joints [75.138, -16.645, 80.833, 0, 25.812, 75.138]
  MoveC 3014 to (57.96, 25.7, -4.5) mm, rotated rx 180 ry 0 rz 90 deg; joints [75.151, -16.643, 80.825, 0, 25.818, 75.151] to (58.06, 26.11, -4.5) mm, rotated rx 180 ry 0 rz 90 deg; joints [75.165, -16.643, 80.826, 0, 25.817, 75.165]
  MoveL 3015 to (58.11, 26.45, -4.5) mm, rotated rx 180 ry 0 rz 90 deg; joints [75.176, -16.644, 80.829, 0, 25.815, 75.176]
  MoveC 3016 to (57.58, 29.82, -4.5) mm, rotated rx -180 ry 0 rz 90 deg; joints [75.279, -16.674, 80.935, 0, 25.739, 75.279] to (55.36, 32.41, -4.5) mm, rotated rx 180 ry 0 rz 90 deg; joints [75.343, -16.734, 81.149, 0, 25.584, 75.343]
  MoveC 3017 to (54.55, 32.79, -4.5) mm, rotated rx 180 ry 0 rz 90 deg; joints [75.348, -16.753, 81.217, 0, 25.536, 75.348] to (53.67, 32.9, -4.5) mm, rotated rx 180 ry 0 rz 90 deg; joints [75.344, -16.772, 81.284, 0, 25.487, 75.344]
  MoveL 3018 to (13.74, 31.82, -4.5) mm, rotated rx -180 ry 0 rz 90 deg; joints [74.97, -17.553, 84.168, 0, 23.385, 74.97]
  MoveL 3019 to (7.52, 31.64, -4.5) mm, rotated rx 180 ry 0 rz 90 deg; joints [74.91, -17.667, 84.609, 0, 23.059, 74.91]
  MoveC 3020 to (3.6, 29.53, -4.5) mm, rotated rx 180 ry 0 rz 90 deg; joints [74.806, -17.729, 84.847, 0, 22.882, 74.806] to (3.08, 25.11, -4.5) mm, rotated rx -180 ry 0 rz 90 deg; joints [74.658, -17.717, 84.798, 0, 22.918, 74.658]
  MoveL 3021 to (9.27, 8.05, -4.5) mm, rotated rx -180 ry 0 rz 90 deg; joints [74.161, -17.513, 84.019, 0, 23.495, 74.161]
  MoveC 3022 to (9.89, 6.94, -4.5) mm, rotated rx 180 ry 0 rz 90 deg; joints [74.131, -17.496, 83.952, 0, 23.544, 74.131] to (10.77, 6.02, -4.5) mm, rotated rx 180 ry 0 rz 90 deg; joints [74.109, -17.474, 83.87, 0, 23.604, 74.109]
  MoveL 3023 to (27.64, -7.11, -4.5) mm, rotated rx 180 ry 0 rz 90 deg; joints [73.844, -17.075, 82.384, 0, 24.691, 73.844]
  MoveL 3024 to (27.96, -7.36, -4.5) mm, rotated rx -180 ry 0 rz 90 deg; joints [73.839, -17.067, 82.356, 0, 24.712, 73.839]
  MoveC 3025 to (31.37, -8.44, -4.5) mm, rotated rx 180 ry 0 rz 90 deg; joints [73.836, -16.993, 82.084, 0, 24.909, 73.836] to (34.59, -6.85, -4.5) mm, rotated rx -180 ry 0 rz 90 deg; joints [73.916, -16.938, 81.883, 0, 25.054, 73.916]
  MoveL 3026 to (35.16, -6.16, -4.5) mm, rotated rx -180 ry 0 rz 90 deg; joints [73.943, -16.93, 81.856, 0, 25.074, 73.943]
  MoveL 3027 to (46.2, 9.22, -4.5) mm, rotated rx 180 ry 0 rz 90 deg; joints [74.529, -16.794, 81.365, 0, 25.429, 74.529]
  MoveL 3028 to (40.07, 13.62, -4.5) mm, rotated rx -180 ry 0 rz 90 deg; joints [74.615, -16.944, 81.905, 0, 25.039, 74.615]
  MoveL 3029 to (40.07, 13.62, -1.5) mm, rotated rx 180 ry 0 rz 90 deg; joints [74.615, -17.096, 82.006, 0, 25.09, 74.615]
  Establecer velocidad (1000.0 mm/s)
  MoveL 3030 to (40.07, 13.62, 10) mm, rotated rx 180 ry 0 rz 90 deg; joints [74.615, -17.677, 82.39, 0, 25.287, 74.615]
  Establecer velocidad (66.7 mm/s)
  MoveL 3031 to (25.29, 68.28, 10) mm, rotated rx -180 ry 0 rz 90 deg; joints [76.251, -18.251, 84.495, 0, 23.756, 76.251]
  MoveL 3032 to (25.29, 68.28, -1.25) mm, rotated rx -180 ry 0 rz 90 deg; joints [76.251, -17.677, 84.12, 0, 23.557, 76.251]
  MoveL 3033 to (25.49, 69.78, -1.66) mm, rotated rx 180 ry 0 rz 90 deg; joints [76.301, -17.66, 84.118, 0, 23.541, 76.301]
  MoveL 3034 to (25.32, 71.29, -2.06) mm, rotated rx 180 ry 0 rz 90 deg; joints [76.349, -17.649, 84.143, 0, 23.506, 76.349]
  MoveL 3035 to (24.83, 72.73, -2.47) mm, rotated rx -180 ry 0 rz 90 deg; joints [76.392, -17.644, 84.19, 0, 23.454, 76.392]
  MoveL 3036 to (24.02, 74.02, -2.88) mm, rotated rx 180 ry 0 rz 90 deg; joints [76.428, -17.645, 84.257, 0, 23.388, 76.428]
  MoveL 3037 to (22.95, 75.1, -3.28) mm, rotated rx 180 ry 0 rz 90 deg; joints [76.455, -17.649, 84.339, 0, 23.31, 76.455]
  MoveL 3038 to (21.67, 75.92, -3.69) mm, rotated rx -180 ry 0 rz 90 deg; joints [76.471, -17.656, 84.431, 0, 23.224, 76.471]
  MoveL 3039 to (20.24, 76.43, -4.09) mm, rotated rx -180 ry 0 rz 90 deg; joints [76.477, -17.664, 84.529, 0, 23.135, 76.477]
  MoveL 3040 to (18.74, 76.58, -4.5) mm, rotated rx -180 ry 0 rz 90 deg; joints [76.47, -17.672, 84.626, 0, 23.046, 76.47]
  MoveL 3041 to (-29.85, 77.07, -4.5) mm, rotated rx 180 ry 0 rz 90 deg; joints [76.093, -18.521, 88.05, 0, 20.471, 76.093]
  MoveC 3042 to (-31.51, 77.04, -4.5) mm, rotated rx -180 ry 0 rz 90 deg; joints [76.078, -18.547, 88.164, 0, 20.384, 76.078] to (-33.17, 76.89, -4.5) mm, rotated rx -180 ry 0 rz 90 deg; joints [76.059, -18.574, 88.275, 0, 20.298, 76.059]
  MoveC 3043 to (-36.21, 73.17, -4.5) mm, rotated rx 180 ry 0 rz 90 deg; joints [75.908, -18.608, 88.42, 0, 20.187, 75.908] to (-35.54, 68.42, -4.5) mm, rotated rx 180 ry 0 rz 90 deg; joints [75.753, -18.577, 88.292, 0, 20.286, 75.753]
  MoveL 3044 to (-34.54, 67.76, -4.5) mm, rotated rx 180 ry 0 rz 90 deg; joints [75.74, -18.559, 88.212, 0, 20.347, 75.74]
  MoveL 3045 to (-11.83, 53.35, -4.5) mm, rotated rx -180 ry 0 rz 90 deg; joints [75.454, -18.117, 86.379, 0, 21.737, 75.454]
  MoveC 3046 to (-9.48, 52.34, -4.5) mm, rotated rx 180 ry 0 rz 90 deg; joints [75.44, -18.071, 86.196, 0, 21.875, 75.44] to (-6.93, 52.12, -4.5) mm, rotated rx 180 ry 0 rz 90 deg; joints [75.455, -18.025, 86.014, 0, 22.012, 75.455]
  MoveL 3047 to (59.23, 56.96, -4.5) mm, rotated rx 180 ry 0 rz 90 deg; joints [76.155, -16.783, 81.325, 0, 25.458, 76.155]
  MoveL 3048 to (70.6, 57.89, -4.5) mm, rotated rx 180 ry 0 rz 90 deg; joints [76.273, -16.549, 80.494, 0, 26.055, 76.273]
  MoveC 3049 to (73.46, 59.18, -4.5) mm, rotated rx 180 ry 0 rz 90 deg; joints [76.336, -16.495, 80.303, 0, 26.192, 76.336] to (74.69, 62.07, -4.5) mm, rotated rx 180 ry 0 rz 90 deg; joints [76.437, -16.483, 80.263, 0, 26.22, 76.437]
  MoveL 3050 to (74.68, 71.35, -4.5) mm, rotated rx 180 ry 0 rz 90 deg; joints [76.731, -16.531, 80.43, 0, 26.101, 76.731]
  MoveC 3051 to (73.51, 74.26, -4.5) mm, rotated rx 180 ry 0 rz 90 deg; joints [76.815, -16.57, 80.57, 0, 26.001, 76.815] to (70.63, 75.53, -4.5) mm, rotated rx 180 ry 0 rz 90 deg; joints [76.834, -16.638, 80.807, 0, 25.831, 76.834]
  MoveC 3052 to (45.03, 76.19, -4.5) mm, rotated rx 180 ry 0 rz 90 deg; joints [76.662, -17.165, 82.714, 0, 24.451, 76.662] to (19.43, 76.58, -4.5) mm, rotated rx -180 ry 0 rz 90 deg; joints [76.475, -17.659, 84.577, 0, 23.083, 76.475]
  MoveL 3053 to (18.74, 76.58, -4.5) mm, rotated rx -180 ry 0 rz 90 deg; joints [76.47, -17.672, 84.626, 0, 23.046, 76.47]
  MoveL 3054 to (18.66, 69.03, -4.5) mm, rotated rx 180 ry 0 rz 90 deg; joints [76.223, -17.639, 84.5, 0, 23.139, 76.223]
  MoveL 3055 to (18.66, 69.03, -1.5) mm, rotated rx -180 ry 0 rz 90 deg; joints [76.223, -17.793, 84.602, 0, 23.191, 76.223]
  Establecer velocidad (1000.0 mm/s)
  MoveL 3056 to (18.66, 69.03, 10) mm, rotated rx -180 ry 0 rz 90 deg; joints [76.223, -18.38, 84.985, 0, 23.396, 76.223]
  Establecer velocidad (66.7 mm/s)
  MoveL 3057 to (25.28, 67.98, 10) mm, rotated rx -180 ry 0 rz 90 deg; joints [76.241, -18.25, 84.49, 0, 23.759, 76.241]
  MoveL 3058 to (25.28, 67.98, -1.5) mm, rotated rx -180 ry 0 rz 90 deg; joints [76.241, -17.663, 84.107, 0, 23.556, 76.241]
  MoveL 3059 to (25.48, 69.48, -1.9) mm, rotated rx 180 ry 0 rz 90 deg; joints [76.292, -17.646, 84.105, 0, 23.54, 76.292]
  MoveL 3060 to (25.32, 70.99, -2.31) mm, rotated rx 180 ry 0 rz 90 deg; joints [76.339, -17.635, 84.13, 0, 23.505, 76.339]
  MoveL 3061 to (24.82, 72.43, -2.72) mm, rotated rx -180 ry 0 rz 90 deg; joints [76.382, -17.63, 84.177, 0, 23.453, 76.382]
  MoveL 3062 to (24.02, 73.72, -3.12) mm, rotated rx 180 ry 0 rz 90 deg; joints [76.418, -17.631, 84.244, 0, 23.387, 76.418]
  MoveL 3063 to (22.95, 74.8, -3.53) mm, rotated rx 180 ry 0 rz 90 deg; joints [76.445, -17.635, 84.326, 0, 23.309, 76.445]
  MoveL 3064 to (21.67, 75.62, -3.94) mm, rotated rx -180 ry 0 rz 90 deg; joints [76.462, -17.642, 84.418, 0, 23.224, 76.462]
  MoveL 3065 to (20.24, 76.13, -4.34) mm, rotated rx 180 ry 0 rz 90 deg; joints [76.467, -17.65, 84.516, 0, 23.134, 76.467]
  MoveL 3066 to (18.73, 76.29, -4.75) mm, rotated rx 180 ry 0 rz 90 deg; joints [76.46, -17.658, 84.613, 0, 23.045, 76.46]
  MoveL 3067 to (-28.9, 76.8, -4.75) mm, rotated rx -180 ry 0 rz 90 deg; joints [76.091, -18.491, 87.971, 0, 20.52, 76.091]
  MoveL 3068 to (-29.85, 76.81, -4.75) mm, rotated rx 180 ry 0 rz 90 deg; joints [76.084, -18.507, 88.037, 0, 20.47, 76.084]
  MoveC 3069 to (-31.21, 76.78, -4.75) mm, rotated rx -180 ry 0 rz 90 deg; joints [76.072, -18.529, 88.13, 0, 20.398, 76.072] to (-32.57, 76.68, -4.75) mm, rotated rx -180 ry 0 rz 90 deg; joints [76.057, -18.55, 88.222, 0, 20.328, 76.057]
  MoveC 3070 to (-35.55, 73.03, -4.75) mm, rotated rx -180 ry 0 rz 90 deg; joints [75.909, -18.583, 88.364, 0, 20.219, 75.909] to (-34.97, 68.36, -4.75) mm, rotated rx 180 ry 0 rz 90 deg; joints [75.756, -18.555, 88.243, 0, 20.312, 75.756]
  MoveL 3071 to (-33.64, 67.48, -4.75) mm, rotated rx 180 ry 0 rz 90 deg; joints [75.738, -18.53, 88.137, 0, 20.393, 75.738]
  MoveL 3072 to (-13.13, 54.49, -4.75) mm, rotated rx 180 ry 0 rz 90 deg; joints [75.48, -18.131, 86.483, 0, 21.648, 75.48]
  MoveL 3073 to (-11.85, 53.68, -4.75) mm, rotated rx -180 ry 0 rz 90 deg; joints [75.464, -18.106, 86.379, 0, 21.727, 75.464]
  MoveC 3074 to (-9.58, 52.65, -4.75) mm, rotated rx 180 ry 0 rz 90 deg; joints [75.45, -18.062, 86.201, 0, 21.86, 75.45] to (-7.11, 52.38, -4.75) mm, rotated rx 180 ry 0 rz 90 deg; joints [75.462, -18.017, 86.023, 0, 21.994, 75.462]
  MoveL 3075 to (53.54, 56.82, -4.75) mm, rotated rx 180 ry 0 rz 90 deg; joints [76.105, -16.887, 81.735, 0, 25.152, 76.105]
  MoveL 3076 to (69.65, 58.16, -4.75) mm, rotated rx -180 ry 0 rz 90 deg; joints [76.274, -16.558, 80.561, 0, 25.997, 76.274]
  MoveL 3077 to (70.59, 58.25, -4.75) mm, rotated rx 180 ry 0 rz 90 deg; joints [76.284, -16.538, 80.492, 0, 26.046, 76.284]
  MoveC 3078 to (73.29, 59.61, -4.75) mm, rotated rx 180 ry 0 rz 90 deg; joints [76.348, -16.488, 80.315, 0, 26.173, 76.348] to (74.37, 62.42, -4.75) mm, rotated rx -180 ry 0 rz 90 deg; joints [76.445, -16.479, 80.285, 0, 26.195, 76.445]
  MoveL 3079 to (74.37, 71.13, -4.75) mm, rotated rx 180 ry 0 rz 90 deg; joints [76.722, -16.524, 80.441, 0, 26.083, 76.722]
  MoveC 3080 to (73.23, 73.95, -4.75) mm, rotated rx 180 ry 0 rz 90 deg; joints [76.803, -16.562, 80.577, 0, 25.986, 76.803] to (70.44, 75.19, -4.75) mm, rotated rx -180 ry 0 rz 90 deg; joints [76.822, -16.627, 80.807, 0, 25.82, 76.822]
  MoveC 3081 to (49.2, 75.82, -4.75) mm, rotated rx 180 ry 0 rz 90 deg; joints [76.682, -17.068, 82.394, 0, 24.674, 76.682] to (27.96, 76.19, -4.75) mm, rotated rx 180 ry 0 rz 90 deg; joints [76.53, -17.484, 83.948, 0, 23.536, 76.53]
  MoveL 3082 to (18.73, 76.29, -4.75) mm, rotated rx 180 ry 0 rz 90 deg; joints [76.46, -17.658, 84.613, 0, 23.045, 76.46]
  MoveL 3083 to (18.65, 68.74, -4.75) mm, rotated rx 180 ry 0 rz 90 deg; joints [76.213, -17.625, 84.487, 0, 23.138, 76.213]
  MoveL 3084 to (18.65, 68.74, -1.75) mm, rotated rx 180 ry 0 rz 90 deg; joints [76.213, -17.779, 84.589, 0, 23.19, 76.213]
  Establecer velocidad (1000.0 mm/s)
  MoveL 3085 to (18.65, 68.74, 10) mm, rotated rx 180 ry 0 rz 90 deg; joints [76.213, -18.379, 84.98, 0, 23.399, 76.213]
  Establecer velocidad (66.7 mm/s)
  MoveL 3086 to (37.6, 23.98, 10) mm, rotated rx -180 ry 0 rz 90 deg; joints [74.924, -17.785, 82.777, 0, 25.008, 74.924]
  MoveL 3087 to (37.6, 23.98, -1.5) mm, rotated rx 180 ry 0 rz 90 deg; joints [74.924, -17.202, 82.393, 0, 24.809, 74.924]
  MoveL 3088 to (37.74, 25.48, -1.9) mm, rotated rx 180 ry 0 rz 90 deg; joints [74.973, -17.187, 82.398, 0, 24.789, 74.973]
  MoveL 3089 to (37.52, 26.99, -2.31) mm, rotated rx 180 ry 0 rz 90 deg; joints [75.019, -17.179, 82.43, 0, 24.749, 75.019]
  MoveL 3090 to (36.97, 28.4, -2.72) mm, rotated rx -180 ry 0 rz 90 deg; joints [75.06, -17.177, 82.484, 0, 24.692, 75.06]
  MoveL 3091 to (36.12, 29.66, -3.12) mm, rotated rx -180 ry 0 rz 90 deg; joints [75.093, -17.18, 82.557, 0, 24.623, 75.093]
  MoveL 3092 to (35.01, 30.7, -3.53) mm, rotated rx 180 ry 0 rz 90 deg; joints [75.117, -17.186, 82.644, 0, 24.542, 75.117]
  MoveL 3093 to (33.7, 31.47, -3.94) mm, rotated rx -180 ry 0 rz 90 deg; joints [75.13, -17.196, 82.741, 0, 24.455, 75.13]
  MoveL 3094 to (32.25, 31.93, -4.34) mm, rotated rx 180 ry 0 rz 90 deg; joints [75.133, -17.206, 82.841, 0, 24.365, 75.133]
  MoveL 3095 to (30.74, 32.03, -4.75) mm, rotated rx -180 ry 0 rz 90 deg; joints [75.123, -17.215, 82.939, 0, 24.276, 75.123]
  MoveL 3096 to (8.05, 31.41, -4.75) mm, rotated rx 180 ry 0 rz 90 deg; joints [74.907, -17.644, 84.558, 0, 23.086, 74.907]
  MoveL 3097 to (7.55, 31.38, -4.75) mm, rotated rx 180 ry 0 rz 90 deg; joints [74.901, -17.653, 84.593, 0, 23.06, 74.901]
  MoveC 3098 to (3.87, 29.31, -4.75) mm, rotated rx -180 ry 0 rz 90 deg; joints [74.801, -17.71, 84.815, 0, 22.896, 74.801] to (3.37, 25.11, -4.75) mm, rotated rx 180 ry 0 rz 90 deg; joints [74.66, -17.698, 84.769, 0, 22.93, 74.66]
  MoveL 3099 to (9.5, 8.22, -4.75) mm, rotated rx -180 ry 0 rz 90 deg; joints [74.169, -17.497, 83.997, 0, 23.5, 74.169]
  MoveC 3100 to (10.09, 7.12, -4.75) mm, rotated rx 180 ry 0 rz 90 deg; joints [74.138, -17.48, 83.933, 0, 23.547, 74.138] to (10.96, 6.22, -4.75) mm, rotated rx 180 ry 0 rz 90 deg; joints [74.118, -17.459, 83.853, 0, 23.607, 74.118]
  MoveL 3101 to (25.64, -5.21, -4.75) mm, rotated rx 180 ry 0 rz 90 deg; joints [73.886, -17.113, 82.56, 0, 24.553, 73.886]
  MoveL 3102 to (28.14, -7.15, -4.75) mm, rotated rx 180 ry 0 rz 90 deg; joints [73.847, -17.052, 82.338, 0, 24.714, 73.847]
  MoveC 3103 to (31.5, -8.1, -4.75) mm, rotated rx 180 ry 0 rz 90 deg; joints [73.848, -16.98, 82.074, 0, 24.906, 73.848] to (34.58, -6.45, -4.75) mm, rotated rx -180 ry 0 rz 90 deg; joints [73.929, -16.928, 81.884, 0, 25.044, 73.929]
  MoveL 3104 to (34.82, -6.16, -4.75) mm, rotated rx 180 ry 0 rz 90 deg; joints [73.94, -16.925, 81.873, 0, 25.052, 73.94]
  MoveL 3105 to (57.33, 25.22, -4.75) mm, rotated rx 180 ry 0 rz 90 deg; joints [75.131, -16.641, 80.854, 0, 25.787, 75.131]
  MoveL 3106 to (57.48, 25.46, -4.75) mm, rotated rx 180 ry 0 rz 90 deg; joints [75.14, -16.639, 80.848, 0, 25.791, 75.14]
  MoveC 3107 to (57.03, 29.7, -4.75) mm, rotated rx -180 ry 0 rz 90 deg; joints [75.27, -16.672, 80.964, 0, 25.708, 75.27] to (53.93, 32.61, -4.75) mm, rotated rx 180 ry 0 rz 90 deg; joints [75.337, -16.752, 81.251, 0, 25.501, 75.337]
  MoveL 3108 to (46.91, 32.47, -4.75) mm, rotated rx -180 ry 0 rz 90 deg; joints [75.274, -16.895, 81.766, 0, 25.129, 75.274]
  MoveL 3109 to (30.74, 32.03, -4.75) mm, rotated rx -180 ry 0 rz 90 deg; joints [75.123, -17.215, 82.939, 0, 24.276, 75.123]
  MoveL 3110 to (30.94, 24.48, -4.75) mm, rotated rx 180 ry 0 rz 90 deg; joints [74.883, -17.172, 82.777, 0, 24.394, 74.883]
  MoveL 3111 to (30.94, 24.48, -1.75) mm, rotated rx -180 ry 0 rz 90 deg; joints [74.883, -17.324, 82.879, 0, 24.445, 74.883]
  Establecer velocidad (1000.0 mm/s)
  MoveL 3112 to (30.94, 24.48, 10) mm, rotated rx -180 ry 0 rz 90 deg; joints [74.883, -17.921, 83.271, 0, 24.65, 74.883]
  Establecer velocidad (66.7 mm/s)
  MoveL 3113 to (66.68, -31.06, 10) mm, rotated rx 180 ry 0 rz 90 deg; joints [73.452, -16.84, 79.468, 0, 27.371, 73.452]
  MoveL 3114 to (66.68, -31.06, -1.5) mm, rotated rx -180 ry 0 rz 90 deg; joints [73.452, -16.264, 79.082, 0, 27.182, 73.452]
  MoveL 3115 to (68.18, -31.25, -1.91) mm, rotated rx -180 ry 0 rz 90 deg; joints [73.46, -16.209, 78.951, 0, 27.258, 73.46]
  MoveL 3116 to (69.69, -31.07, -2.31) mm, rotated rx -180 ry 0 rz 90 deg; joints [73.48, -16.156, 78.827, 0, 27.329, 73.48]
  MoveL 3117 to (71.12, -30.56, -2.72) mm, rotated rx 180 ry 0 rz 90 deg; joints [73.509, -16.108, 78.717, 0, 27.391, 73.509]
  MoveL 3118 to (72.41, -29.74, -3.12) mm, rotated rx -180 ry 0 rz 90 deg; joints [73.545, -16.064, 78.624, 0, 27.44, 73.545]
  MoveL 3119 to (73.47, -28.66, -3.53) mm, rotated rx -180 ry 0 rz 90 deg; joints [73.588, -16.027, 78.553, 0, 27.473, 73.588]
  MoveL 3120 to (74.28, -27.37, -3.94) mm, rotated rx -180 ry 0 rz 90 deg; joints [73.636, -15.997, 78.507, 0, 27.49, 73.636]
  MoveL 3121 to (74.78, -25.94, -4.34) mm, rotated rx 180 ry 0 rz 90 deg; joints [73.684, -15.975, 78.488, 0, 27.487, 73.684]
  MoveL 3122 to (74.92, -24.43, -4.75) mm, rotated rx 180 ry 0 rz 90 deg; joints [73.732, -15.961, 78.497, 0, 27.465, 73.732]
  MoveL 3123 to (74.92, -8.05, -4.75) mm, rotated rx 180 ry 0 rz 90 deg; joints [74.239, -16.066, 78.852, 0, 27.213, 74.239]
  MoveL 3124 to (74.91, -6.63, -4.75) mm, rotated rx -180 ry 0 rz 90 deg; joints [74.283, -16.075, 78.883, 0, 27.192, 74.283]
  MoveC 3125 to (72.79, -3.88, -4.75) mm, rotated rx 180 ry 0 rz 90 deg; joints [74.35, -16.139, 79.102, 0, 27.037, 74.35] to (69.65, -2.37, -4.75) mm, rotated rx -180 ry 0 rz 90 deg; joints [74.37, -16.217, 79.37, 0, 26.846, 74.37]
  MoveC 3126 to (68.21, -2.29, -4.75) mm, rotated rx -180 ry 0 rz 90 deg; joints [74.36, -16.249, 79.481, 0, 26.768, 74.36] to (66.81, -2.67, -4.75) mm, rotated rx -180 ry 0 rz 90 deg; joints [74.336, -16.277, 79.578, 0, 26.699, 74.336]
  MoveL 3127 to (51.65, -23.45, -4.75) mm, rotated rx -180 ry 0 rz 90 deg; joints [73.55, -16.473, 80.263, 0, 26.21, 73.55]
  MoveC 3128 to (50.81, -26.22, -4.75) mm, rotated rx -180 ry 0 rz 90 deg; joints [73.456, -16.473, 80.264, 0, 26.21, 73.456] to (51.91, -28.9, -4.75) mm, rotated rx -180 ry 0 rz 90 deg; joints [73.383, -16.433, 80.124, 0, 26.31, 73.383]
  MoveL 3129 to (53.59, -30.8, -4.75) mm, rotated rx 180 ry 0 rz 90 deg; joints [73.339, -16.386, 79.956, 0, 26.429, 73.339]
  MoveL 3130 to (65.32, -44.07, -4.75) mm, rotated rx 180 ry 0 rz 90 deg; joints [73.038, -16.044, 78.779, 0, 27.265, 73.038]
  MoveL 3131 to (67.23, -46.21, -4.75) mm, rotated rx -180 ry 0 rz 90 deg; joints [72.99, -15.988, 78.585, 0, 27.402, 72.99]
  MoveC 3132 to (69.43, -46.54, -4.75) mm, rotated rx -180 ry 0 rz 90 deg; joints [73, -15.936, 78.412, 0, 27.524, 73] to (71.55, -45.88, -4.75) mm, rotated rx 180 ry 0 rz 90 deg; joints [73.04, -15.894, 78.267, 0, 27.627, 73.04]
  MoveL 3133 to (72.07, -45.56, -4.75) mm, rotated rx 180 ry 0 rz 90 deg; joints [73.055, -15.884, 78.235, 0, 27.649, 73.055]
  MoveC 3134 to (73.76, -44.12, -4.75) mm, rotated rx -180 ry 0 rz 90 deg; joints [73.115, -15.856, 78.14, 0, 27.716, 73.115] to (74.91, -42.22, -4.75) mm, rotated rx 180 ry 0 rz 90 deg; joints [73.184, -15.843, 78.096, 0, 27.747, 73.184]
  MoveL 3135 to (74.92, -24.43, -4.75) mm, rotated rx 180 ry 0 rz 90 deg; joints [73.732, -15.961, 78.497, 0, 27.465, 73.732]
  MoveL 3136 to (67.37, -24.42, -4.75) mm, rotated rx -180 ry 0 rz 90 deg; joints [73.664, -16.128, 79.067, 0, 27.062, 73.664]
  MoveL 3137 to (67.37, -24.42, -1.75) mm, rotated rx 180 ry 0 rz 90 deg; joints [73.664, -16.279, 79.169, 0, 27.11, 73.664]
  Establecer velocidad (1000.0 mm/s)
  MoveL 3138 to (67.37, -24.42, 10) mm, rotated rx 180 ry 0 rz 90 deg; joints [73.664, -16.868, 79.564, 0, 27.304, 73.664]
  Establecer velocidad (66.7 mm/s)
  MoveL 3139 to (18.15, -68.23, 10) mm, rotated rx -180 ry 0 rz 90 deg; joints [71.823, -17.621, 82.189, 0, 25.432, 71.823]
  MoveL 3140 to (18.15, -68.23, -1.5) mm, rotated rx 180 ry 0 rz 90 deg; joints [71.823, -17.04, 81.804, 0, 25.235, 71.823]
  MoveL 3141 to (17.99, -69.74, -1.91) mm, rotated rx 180 ry 0 rz 90 deg; joints [71.774, -17.013, 81.767, 0, 25.246, 71.774]
  MoveL 3142 to (18.18, -71.25, -2.31) mm, rotated rx -180 ry 0 rz 90 deg; joints [71.729, -16.978, 81.703, 0, 25.275, 71.729]
  MoveL 3143 to (18.71, -72.67, -2.72) mm, rotated rx -180 ry 0 rz 90 deg; joints [71.69, -16.938, 81.617, 0, 25.321, 71.69]
  MoveL 3144 to (19.54, -73.95, -3.12) mm, rotated rx 180 ry 0 rz 90 deg; joints [71.659, -16.892, 81.513, 0, 25.379, 71.659]
  MoveL 3145 to (20.63, -75, -3.53) mm, rotated rx 180 ry 0 rz 90 deg; joints [71.637, -16.842, 81.395, 0, 25.448, 71.637]
  MoveL 3146 to (21.93, -75.8, -3.94) mm, rotated rx 180 ry 0 rz 90 deg; joints [71.626, -16.79, 81.267, 0, 25.523, 71.626]
  MoveL 3147 to (23.37, -76.28, -4.34) mm, rotated rx 180 ry 0 rz 90 deg; joints [71.626, -16.737, 81.137, 0, 25.6, 71.626]
  MoveL 3148 to (24.88, -76.4, -4.75) mm, rotated rx 180 ry 0 rz 90 deg; joints [71.637, -16.685, 81.011, 0, 25.674, 71.637]
  MoveL 3149 to (52.59, -76.11, -4.75) mm, rotated rx -180 ry 0 rz 90 deg; joints [71.928, -16.102, 78.975, 0, 27.127, 71.928]
  MoveL 3150 to (53.11, -76.09, -4.75) mm, rotated rx 180 ry 0 rz 90 deg; joints [71.934, -16.091, 78.937, 0, 27.154, 71.934]
  MoveC 3151 to (56.1, -72.91, -4.75) mm, rotated rx -180 ry 0 rz 90 deg; joints [72.062, -16.048, 78.79, 0, 27.257, 72.062] to (56.24, -68.54, -4.75) mm, rotated rx 180 ry 0 rz 90 deg; joints [72.197, -16.076, 78.886, 0, 27.19, 72.197]
  MoveL 3152 to (56.12, -68.38, -4.75) mm, rotated rx -180 ry 0 rz 90 deg; joints [72.201, -16.079, 78.898, 0, 27.181, 72.201]
  MoveL 3153 to (27.74, -35.54, -4.75) mm, rotated rx 180 ry 0 rz 90 deg; joints [72.945, -16.891, 81.752, 0, 25.139, 72.945]
  MoveL 3154 to (27.01, -34.73, -4.75) mm, rotated rx -180 ry 0 rz 90 deg; joints [72.964, -16.911, 81.823, 0, 25.088, 72.964]
  MoveL 3155 to (26.85, -34.59, -4.75) mm, rotated rx 180 ry 0 rz 90 deg; joints [72.967, -16.915, 81.838, 0, 25.077, 72.967]
  MoveL 3156 to (12.79, -23.33, -4.75) mm, rotated rx -180 ry 0 rz 90 deg; joints [73.188, -17.259, 83.1, 0, 24.159, 73.188]
  MoveL 3157 to (11.85, -22.61, -4.75) mm, rotated rx -180 ry 0 rz 90 deg; joints [73.202, -17.281, 83.184, 0, 24.098, 73.202]
  MoveC 3158 to (8.39, -21.66, -4.75) mm, rotated rx 180 ry 0 rz 90 deg; joints [73.199, -17.353, 83.451, 0, 23.901, 73.199] to (5.21, -23.31, -4.75) mm, rotated rx -180 ry 0 rz 90 deg; joints [73.115, -17.404, 83.643, 0, 23.761, 73.115]
  MoveC 3159 to (4.69, -24.17, -4.75) mm, rotated rx 180 ry 0 rz 90 deg; joints [73.083, -17.409, 83.662, 0, 23.747, 73.083] to (4.36, -25.11, -4.75) mm, rotated rx -180 ry 0 rz 90 deg; joints [73.049, -17.409, 83.665, 0, 23.745, 73.049]
  MoveL 3160 to (-7.74, -70.6, -4.75) mm, rotated rx -180 ry 0 rz 90 deg; joints [71.478, -17.363, 83.49, 0, 23.873, 71.478]
  MoveC 3161 to (-7.03, -74.71, -4.75) mm, rotated rx 180 ry 0 rz 90 deg; joints [71.356, -17.324, 83.343, 0, 23.981, 71.356] to (-3.35, -76.66, -4.75) mm, rotated rx -180 ry 0 rz 90 deg; joints [71.334, -17.241, 83.035, 0, 24.207, 71.334]
  MoveC 3162 to (-2.27, -76.68, -4.75) mm, rotated rx -180 ry 0 rz 90 deg; joints [71.344, -17.221, 82.958, 0, 24.263, 71.344] to (-1.2, -76.68, -4.75) mm, rotated rx 180 ry 0 rz 90 deg; joints [71.356, -17.2, 82.881, 0, 24.319, 71.356]
  MoveL 3163 to (24.88, -76.4, -4.75) mm, rotated rx 180 ry 0 rz 90 deg; joints [71.637, -16.685, 81.011, 0, 25.674, 71.637]
  MoveL 3164 to (24.8, -68.85, -4.75) mm, rotated rx 180 ry 0 rz 90 deg; joints [71.872, -16.737, 81.197, 0, 25.54, 71.872]
  MoveL 3165 to (24.8, -68.85, -1.75) mm, rotated rx 180 ry 0 rz 90 deg; joints [71.872, -16.889, 81.299, 0, 25.59, 71.872]
  Establecer velocidad (1000.0 mm/s)
  MoveL 3166 to (24.8, -68.85, 10) mm, rotated rx -180 ry 0 rz 90 deg; joints [71.872, -17.481, 81.692, 0, 25.789, 71.872]
  Establecer velocidad (66.7 mm/s)
  MoveL 3167 to (-32.95, -52.17, 10) mm, rotated rx -180 ry 0 rz 90 deg; joints [71.8, -18.689, 86.175, 0, 22.514, 71.8]
  MoveL 3168 to (-32.95, -52.17, -1.5) mm, rotated rx -180 ry 0 rz 90 deg; joints [71.8, -18.099, 85.792, 0, 22.306, 71.8]
  MoveL 3169 to (-31.54, -52.73, -1.9) mm, rotated rx -180 ry 0 rz 90 deg; joints [71.797, -18.05, 85.668, 0, 22.382, 71.797]
  MoveL 3170 to (-30.03, -52.93, -2.31) mm, rotated rx -180 ry 0 rz 90 deg; joints [71.806, -18.001, 85.546, 0, 22.456, 71.806]
  MoveL 3171 to (-28.52, -52.8, -2.72) mm, rotated rx 180 ry 0 rz 90 deg; joints [71.827, -17.955, 85.43, 0, 22.525, 71.827]
  MoveL 3172 to (-27.07, -52.33, -3.12) mm, rotated rx 180 ry 0 rz 90 deg; joints [71.857, -17.911, 85.326, 0, 22.584, 71.857]
  MoveL 3173 to (-25.77, -51.55, -3.53) mm, rotated rx 180 ry 0 rz 90 deg; joints [71.896, -17.871, 85.239, 0, 22.632, 71.896]
  MoveL 3174 to (-24.66, -50.51, -3.94) mm, rotated rx 180 ry 0 rz 90 deg; joints [71.941, -17.837, 85.173, 0, 22.664, 71.941]
  MoveL 3175 to (-23.82, -49.25, -4.34) mm, rotated rx 180 ry 0 rz 90 deg; joints [71.99, -17.808, 85.129, 0, 22.68, 71.99]
  MoveL 3176 to (-23.3, -47.82, -4.75) mm, rotated rx -180 ry 0 rz 90 deg; joints [72.042, -17.786, 85.111, 0, 22.675, 72.042]
  MoveL 3177 to (-17.03, -23.75, -4.75) mm, rotated rx 180 ry 0 rz 90 deg; joints [72.882, -17.81, 85.205, 0, 22.606, 72.882]
  MoveC 3178 to (-16.76, -22.08, -4.75) mm, rotated rx -180 ry 0 rz 90 deg; joints [72.939, -17.815, 85.221, 0, 22.593, 72.939] to (-16.79, -20.38, -4.75) mm, rotated rx 180 ry 0 rz 90 deg; joints [72.994, -17.825, 85.26, 0, 22.564, 72.994]
  MoveC 3179 to (-18.27, -17.4, -4.75) mm, rotated rx 180 ry 0 rz 90 deg; joints [73.076, -17.867, 85.427, 0, 22.44, 73.076] to (-21.3, -16.05, -4.75) mm, rotated rx 180 ry 0 rz 90 deg; joints [73.09, -17.928, 85.668, 0, 22.26, 73.09]
  MoveC 3180 to (-22.46, -16.04, -4.75) mm, rotated rx -180 ry 0 rz 90 deg; joints [73.078, -17.948, 85.748, 0, 22.2, 73.078] to (-23.6, -16.2, -4.75) mm, rotated rx -180 ry 0 rz 90 deg; joints [73.062, -17.967, 85.824, 0, 22.143, 73.062]
  MoveL 3181 to (-72.74, -26.65, -4.75) mm, rotated rx -180 ry 0 rz 90 deg; joints [72.213, -18.72, 88.956, 0, 19.764, 72.213]
  MoveC 3182 to (-76.08, -28.7, -4.75) mm, rotated rx 180 ry 0 rz 90 deg; joints [72.109, -18.761, 89.136, 0, 19.626, 72.109] to (-77.38, -32.39, -4.75) mm, rotated rx 180 ry 0 rz 90 deg; joints [71.972, -18.763, 89.143, 0, 19.62, 71.972]
  MoveL 3183 to (-77.38, -70.6, -4.75) mm, rotated rx -180 ry 0 rz 90 deg; joints [70.71, -18.564, 88.281, 0, 20.283, 70.71]
  MoveC 3184 to (-77.13, -72.58, -4.75) mm, rotated rx 180 ry 0 rz 90 deg; joints [70.648, -18.549, 88.217, 0, 20.332, 70.648] to (-76.29, -74.39, -4.75) mm, rotated rx -180 ry 0 rz 90 deg; joints [70.598, -18.526, 88.118, 0, 20.408, 70.598]
  MoveC 3185 to (-74.19, -76.11, -4.75) mm, rotated rx 180 ry 0 rz 90 deg; joints [70.566, -18.483, 87.937, 0, 20.546, 70.566] to (-71.55, -76.75, -4.75) mm, rotated rx -180 ry 0 rz 90 deg; joints [70.576, -18.437, 87.744, 0, 20.693, 70.576]
  MoveL 3186 to (-70.6, -76.76, -4.75) mm, rotated rx 180 ry 0 rz 90 deg; joints [70.586, -18.422, 87.68, 0, 20.742, 70.586]
  MoveL 3187 to (-42.17, -76.53, -4.75) mm, rotated rx 180 ry 0 rz 90 deg; joints [70.915, -17.949, 85.752, 0, 22.197, 70.915]
  MoveL 3188 to (-35.54, -76.47, -4.75) mm, rotated rx -180 ry 0 rz 90 deg; joints [70.991, -17.834, 85.296, 0, 22.538, 70.991]
  MoveC 3189 to (-34.08, -76.32, -4.75) mm, rotated rx -180 ry 0 rz 90 deg; joints [71.011, -17.809, 85.199, 0, 22.61, 71.011] to (-32.69, -75.86, -4.75) mm, rotated rx -180 ry 0 rz 90 deg; joints [71.041, -17.787, 85.114, 0, 22.673, 71.041]
  MoveC 3190 to (-30.72, -74.2, -4.75) mm, rotated rx 180 ry 0 rz 90 deg; joints [71.116, -17.762, 85.016, 0, 22.746, 71.116] to (-29.57, -71.88, -4.75) mm, rotated rx -180 ry 0 rz 90 deg; joints [71.203, -17.756, 84.991, 0, 22.765, 71.203]
  MoveL 3191 to (-23.3, -47.82, -4.75) mm, rotated rx -180 ry 0 rz 90 deg; joints [72.042, -17.786, 85.111, 0, 22.675, 72.042]
  MoveL 3192 to (-30.61, -45.92, -4.75) mm, rotated rx 180 ry 0 rz 90 deg; joints [72.027, -17.926, 85.662, 0, 22.264, 72.027]
  MoveL 3193 to (-30.61, -45.92, -1.75) mm, rotated rx 180 ry 0 rz 90 deg; joints [72.027, -18.081, 85.763, 0, 22.317, 72.027]
  Establecer velocidad (1000.0 mm/s)
  MoveL 3194 to (-30.61, -45.92, 10) mm, rotated rx 180 ry 0 rz 90 deg; joints [72.027, -18.684, 86.154, 0, 22.53, 72.027]
  Establecer velocidad (66.7 mm/s)
  MoveL 3195 to (-69.14, 36.17, 10) mm, rotated rx -180 ry 0 rz 90 deg; joints [74.36, -19.724, 90.473, 0, 19.251, 74.36]
  MoveL 3196 to (-69.14, 36.17, -1.5) mm, rotated rx 180 ry 0 rz 90 deg; joints [74.36, -19.121, 90.089, 0, 19.032, 74.36]
  MoveL 3197 to (-70.65, 36.36, -1.91) mm, rotated rx -180 ry 0 rz 90 deg; joints [74.352, -19.123, 90.18, 0, 18.943, 74.352]
  MoveL 3198 to (-72.16, 36.17, -2.31) mm, rotated rx -180 ry 0 rz 90 deg; joints [74.332, -19.124, 90.264, 0, 18.86, 74.332]
  MoveL 3199 to (-73.59, 35.66, -2.72) mm, rotated rx 180 ry 0 rz 90 deg; joints [74.301, -19.121, 90.336, 0, 18.785, 74.301]
  MoveL 3200 to (-74.87, 34.84, -3.12) mm, rotated rx 180 ry 0 rz 90 deg; joints [74.26, -19.115, 90.393, 0, 18.722, 74.26]
  MoveL 3201 to (-75.94, 33.76, -3.53) mm, rotated rx 180 ry 0 rz 90 deg; joints [74.213, -19.105, 90.43, 0, 18.675, 74.213]
  MoveL 3202 to (-76.74, 32.48, -3.94) mm, rotated rx 180 ry 0 rz 90 deg; joints [74.162, -19.09, 90.446, 0, 18.644, 74.162]
  MoveL 3203 to (-77.24, 31.04, -4.34) mm, rotated rx 180 ry 0 rz 90 deg; joints [74.108, -19.07, 90.438, 0, 18.632, 74.108]
  MoveL 3204 to (-77.38, 29.53, -4.75) mm, rotated rx -180 ry 0 rz 90 deg; joints [74.055, -19.045, 90.405, 0, 18.64, 74.055]
  MoveL 3205 to (-77.38, 0.78, -4.75) mm, rotated rx -180 ry 0 rz 90 deg; joints [73.082, -18.92, 89.84, 0, 19.08, 73.082]
  MoveC 3206 to (-77.27, -0.48, -4.75) mm, rotated rx -180 ry 0 rz 90 deg; joints [73.041, -18.913, 89.807, 0, 19.106, 73.041] to (-76.95, -1.7, -4.75) mm, rotated rx 180 ry 0 rz 90 deg; joints [73.003, -18.902, 89.761, 0, 19.142, 73.003]
  MoveC 3207 to (-75.45, -3.89, -4.75) mm, rotated rx -180 ry 0 rz 90 deg; joints [72.945, -18.87, 89.615, 0, 19.255, 72.945] to (-73.05, -5.03, -4.75) mm, rotated rx -180 ry 0 rz 90 deg; joints [72.932, -18.829, 89.432, 0, 19.397, 72.932]
  MoveC 3208 to (-71.35, -5.16, -4.75) mm, rotated rx -180 ry 0 rz 90 deg; joints [72.945, -18.802, 89.315, 0, 19.487, 72.945] to (-69.65, -4.94, -4.75) mm, rotated rx 180 ry 0 rz 90 deg; joints [72.969, -18.777, 89.206, 0, 19.572, 72.969]
  MoveL 3209 to (-20.13, 6.45, -4.75) mm, rotated rx -180 ry 0 rz 90 deg; joints [73.835, -18.024, 86.052, 0, 21.973, 73.835]
  MoveC 3210 to (-17.69, 7.7, -4.75) mm, rotated rx -180 ry 0 rz 90 deg; joints [73.899, -17.988, 85.906, 0, 22.081, 73.899] to (-16.12, 9.95, -4.75) mm, rotated rx 180 ry 0 rz 90 deg; joints [73.987, -17.972, 85.842, 0, 22.13, 73.987]
  MoveC 3211 to (-15.82, 12.02, -4.75) mm, rotated rx -180 ry 0 rz 90 deg; joints [74.058, -17.977, 85.863, 0, 22.114, 74.058] to (-16.2, 14.09, -4.75) mm, rotated rx 180 ry 0 rz 90 deg; joints [74.122, -17.994, 85.93, 0, 22.064, 74.122]
  MoveL 3212 to (-22.98, 33.07, -4.75) mm, rotated rx -180 ry 0 rz 90 deg; joints [74.685, -18.202, 86.772, 0, 21.43, 74.685]
  MoveC 3213 to (-23.95, 34.81, -4.75) mm, rotated rx -180 ry 0 rz 90 deg; joints [74.733, -18.227, 86.872, 0, 21.355, 74.733] to (-25.42, 36.14, -4.75) mm, rotated rx 180 ry 0 rz 90 deg; joints [74.764, -18.258, 86.999, 0, 21.259, 74.764]
  MoveL 3214 to (-67.76, 63.31, -4.75) mm, rotated rx 180 ry 0 rz 90 deg; joints [75.298, -19.039, 90.38, 0, 18.659, 75.298]
  MoveC 3215 to (-69.58, 64.22, -4.75) mm, rotated rx 180 ry 0 rz 90 deg; joints [75.313, -19.069, 90.518, 0, 18.551, 75.313] to (-71.55, 64.74, -4.75) mm, rotated rx -180 ry 0 rz 90 deg; joints [75.313, -19.1, 90.659, 0, 18.441, 75.313]
  MoveC 3216 to (-75.01, 64.01, -4.75) mm, rotated rx 180 ry 0 rz 90 deg; joints [75.257, -19.147, 90.877, 0, 18.269, 75.257] to (-77.05, 61.12, -4.75) mm, rotated rx 180 ry 0 rz 90 deg; joints [75.139, -19.165, 90.963, 0, 18.203, 75.139]
  MoveC 3217 to (-77.31, 59.71, -4.75) mm, rotated rx -180 ry 0 rz 90 deg; joints [75.088, -19.163, 90.955, 0, 18.208, 75.088] to (-77.38, 58.28, -4.75) mm, rotated rx -180 ry 0 rz 90 deg; joints [75.038, -19.159, 90.934, 0, 18.225, 75.038]
  MoveL 3218 to (-77.38, 29.53, -4.75) mm, rotated rx -180 ry 0 rz 90 deg; joints [74.055, -19.045, 90.405, 0, 18.64, 74.055]
  MoveL 3219 to (-69.83, 29.53, -4.75) mm, rotated rx -180 ry 0 rz 90 deg; joints [74.128, -18.934, 89.9, 0, 19.033, 74.128]
  MoveL 3220 to (-69.83, 29.53, -1.75) mm, rotated rx -180 ry 0 rz 90 deg; joints [74.128, -19.091, 90.002, 0, 19.089, 74.128]
  Establecer velocidad (1000.0 mm/s)
  MoveL 3221 to (-69.83, 29.53, 10) mm, rotated rx 180 ry 0 rz 90 deg; joints [74.128, -19.706, 90.393, 0, 19.313, 74.128]
  Establecer velocidad (66.7 mm/s)
  MoveL 3222 to (-68.88, 36.17, 10) mm, rotated rx 180 ry 0 rz 90 deg; joints [74.363, -19.72, 90.455, 0, 19.265, 74.363]
  MoveL 3223 to (-68.88, 36.17, -1.75) mm, rotated rx -180 ry 0 rz 90 deg; joints [74.363, -19.104, 90.063, 0, 19.041, 74.363]
  MoveL 3224 to (-70.39, 36.36, -2.16) mm, rotated rx 180 ry 0 rz 90 deg; joints [74.355, -19.106, 90.154, 0, 18.952, 74.355]
  MoveL 3225 to (-71.89, 36.17, -2.56) mm, rotated rx 180 ry 0 rz 90 deg; joints [74.334, -19.107, 90.238, 0, 18.869, 74.334]
  MoveL 3226 to (-73.32, 35.66, -2.97) mm, rotated rx -180 ry 0 rz 90 deg; joints [74.303, -19.104, 90.31, 0, 18.794, 74.303]
  MoveL 3227 to (-74.61, 34.84, -3.38) mm, rotated rx -180 ry 0 rz 90 deg; joints [74.263, -19.098, 90.367, 0, 18.731, 74.263]
  MoveL 3228 to (-75.68, 33.76, -3.78) mm, rotated rx -180 ry 0 rz 90 deg; joints [74.216, -19.088, 90.404, 0, 18.684, 74.216]
  MoveL 3229 to (-76.48, 32.48, -4.19) mm, rotated rx -180 ry 0 rz 90 deg; joints [74.164, -19.073, 90.42, 0, 18.653, 74.164]
  MoveL 3230 to (-76.98, 31.04, -4.59) mm, rotated rx 180 ry 0 rz 90 deg; joints [74.111, -19.053, 90.412, 0, 18.641, 74.111]
  MoveL 3231 to (-77.12, 29.53, -5) mm, rotated rx -180 ry 0 rz 90 deg; joints [74.058, -19.028, 90.379, 0, 18.649, 74.058]
  MoveL 3232 to (-77.12, 1.42, -5) mm, rotated rx 180 ry 0 rz 90 deg; joints [73.107, -18.906, 89.827, 0, 19.079, 73.107]
  MoveL 3233 to (-77.11, 0.47, -5) mm, rotated rx 180 ry 0 rz 90 deg; joints [73.075, -18.902, 89.807, 0, 19.094, 73.075]
  MoveC 3234 to (-76.58, -1.95, -5) mm, rotated rx 180 ry 0 rz 90 deg; joints [72.999, -18.883, 89.722, 0, 19.16, 72.999] to (-75.04, -3.9, -5) mm, rotated rx 180 ry 0 rz 90 deg; joints [72.949, -18.851, 89.579, 0, 19.271, 72.949]
  MoveC 3235 to (-72.65, -4.84, -5) mm, rotated rx 180 ry 0 rz 90 deg; joints [72.942, -18.81, 89.4, 0, 19.41, 72.942] to (-70.08, -4.78, -5) mm, rotated rx -180 ry 0 rz 90 deg; joints [72.971, -18.772, 89.23, 0, 19.542, 72.971]
  MoveL 3236 to (-20.37, 6.66, -5) mm, rotated rx 180 ry 0 rz 90 deg; joints [73.84, -18.017, 86.064, 0, 21.952, 73.84]
  MoveC 3237 to (-18.3, 7.57, -5) mm, rotated rx 180 ry 0 rz 90 deg; joints [73.889, -17.985, 85.938, 0, 22.047, 73.889] to (-16.74, 9.2, -5) mm, rotated rx 180 ry 0 rz 90 deg; joints [73.957, -17.966, 85.862, 0, 22.104, 73.957]
  MoveC 3238 to (-16.09, 11.43, -5) mm, rotated rx -180 ry 0 rz 90 deg; joints [74.036, -17.966, 85.861, 0, 22.105, 74.036] to (-16.37, 13.74, -5) mm, rotated rx 180 ry 0 rz 90 deg; joints [74.109, -17.982, 85.926, 0, 22.056, 74.109]
  MoveL 3239 to (-23.24, 32.99, -5) mm, rotated rx -180 ry 0 rz 90 deg; joints [74.68, -18.193, 86.78, 0, 21.413, 74.68]
  MoveC 3240 to (-24.17, 34.67, -5) mm, rotated rx -180 ry 0 rz 90 deg; joints [74.727, -18.217, 86.877, 0, 21.34, 74.727] to (-25.6, 35.96, -5) mm, rotated rx 180 ry 0 rz 90 deg; joints [74.757, -18.247, 87, 0, 21.247, 74.757]
  MoveL 3241 to (-67.76, 62.99, -5) mm, rotated rx -180 ry 0 rz 90 deg; joints [75.287, -19.025, 90.366, 0, 18.659, 75.287]
  MoveC 3242 to (-69.57, 63.94, -5) mm, rotated rx -180 ry 0 rz 90 deg; joints [75.303, -19.055, 90.505, 0, 18.55, 75.303] to (-71.55, 64.49, -5) mm, rotated rx 180 ry 0 rz 90 deg; joints [75.304, -19.086, 90.646, 0, 18.44, 75.304]
  MoveC 3243 to (-74.8, 63.8, -5) mm, rotated rx 180 ry 0 rz 90 deg; joints [75.251, -19.13, 90.852, 0, 18.278, 75.251] to (-76.78, 61.13, -5) mm, rotated rx 180 ry 0 rz 90 deg; joints [75.141, -19.148, 90.936, 0, 18.212, 75.141]
  MoveC 3244 to (-77.04, 59.89, -5) mm, rotated rx -180 ry 0 rz 90 deg; joints [75.097, -19.147, 90.931, 0, 18.216, 75.097] to (-77.12, 58.63, -5) mm, rotated rx -180 ry 0 rz 90 deg; joints [75.052, -19.143, 90.915, 0, 18.229, 75.052]
  MoveL 3245 to (-77.12, 29.53, -5) mm, rotated rx -180 ry 0 rz 90 deg; joints [74.058, -19.028, 90.379, 0, 18.649, 74.058]
  MoveL 3246 to (-69.57, 29.53, -5) mm, rotated rx 180 ry 0 rz 90 deg; joints [74.131, -18.917, 89.874, 0, 19.042, 74.131]
  MoveL 3247 to (-69.57, 29.53, -2) mm, rotated rx 180 ry 0 rz 90 deg; joints [74.131, -19.074, 89.976, 0, 19.098, 74.131]
  Establecer velocidad (1000.0 mm/s)
  MoveL 3248 to (-69.57, 29.53, 10) mm, rotated rx 180 ry 0 rz 90 deg; joints [74.131, -19.702, 90.376, 0, 19.326, 74.131]
  Establecer velocidad (66.7 mm/s)
  MoveL 3249 to (-39.28, -28.23, 10) mm, rotated rx -180 ry 0 rz 90 deg; joints [72.511, -18.934, 87.144, 0, 21.79, 72.511]
  MoveL 3250 to (-39.28, -28.23, -1.75) mm, rotated rx 180 ry 0 rz 90 deg; joints [72.511, -18.328, 86.753, 0, 21.575, 72.511]
  MoveL 3251 to (-39.42, -26.72, -2.16) mm, rotated rx -180 ry 0 rz 90 deg; joints [72.559, -18.317, 86.781, 0, 21.536, 72.559]
  MoveL 3252 to (-39.91, -25.28, -2.56) mm, rotated rx 180 ry 0 rz 90 deg; joints [72.601, -18.312, 86.832, 0, 21.48, 72.601]
  MoveL 3253 to (-40.71, -23.99, -2.97) mm, rotated rx 180 ry 0 rz 90 deg; joints [72.635, -18.311, 86.901, 0, 21.41, 72.635]
  MoveL 3254 to (-41.77, -22.91, -3.38) mm, rotated rx -180 ry 0 rz 90 deg; joints [72.66, -18.314, 86.984, 0, 21.33, 72.66]
  MoveL 3255 to (-43.05, -22.08, -3.78) mm, rotated rx -180 ry 0 rz 90 deg; joints [72.674, -18.318, 87.075, 0, 21.243, 72.674]
  MoveL 3256 to (-44.48, -21.56, -4.19) mm, rotated rx -180 ry 0 rz 90 deg; joints [72.676, -18.324, 87.17, 0, 21.154, 72.676]
  MoveL 3257 to (-45.99, -21.37, -4.59) mm, rotated rx 180 ry 0 rz 90 deg; joints [72.667, -18.329, 87.264, 0, 21.065, 72.667]
  MoveL 3258 to (-47.49, -21.55, -5) mm, rotated rx -180 ry 0 rz 90 deg; joints [72.646, -18.332, 87.349, 0, 20.982, 72.646]
  MoveL 3259 to (-72.7, -26.92, -5) mm, rotated rx 180 ry 0 rz 90 deg; joints [72.204, -18.705, 88.939, 0, 19.766, 72.204]
  MoveC 3260 to (-75.88, -28.87, -5) mm, rotated rx -180 ry 0 rz 90 deg; joints [72.105, -18.744, 89.11, 0, 19.634, 72.105] to (-77.12, -32.38, -5) mm, rotated rx -180 ry 0 rz 90 deg; joints [71.975, -18.746, 89.117, 0, 19.629, 71.975]
  MoveL 3261 to (-77.12, -71.1, -5) mm, rotated rx 180 ry 0 rz 90 deg; joints [70.696, -18.544, 88.243, 0, 20.301, 70.696]
  MoveC 3262 to (-76.19, -74.08, -5) mm, rotated rx 180 ry 0 rz 90 deg; joints [70.61, -18.513, 88.111, 0, 20.402, 70.61] to (-73.74, -76.01, -5) mm, rotated rx 180 ry 0 rz 90 deg; joints [70.575, -18.463, 87.9, 0, 20.563, 70.575]
  MoveC 3263 to (-72.39, -76.38, -5) mm, rotated rx 180 ry 0 rz 90 deg; joints [70.578, -18.44, 87.801, 0, 20.639, 70.578] to (-70.99, -76.5, -5) mm, rotated rx -180 ry 0 rz 90 deg; joints [70.59, -18.417, 87.705, 0, 20.712, 70.59]
  MoveL 3264 to (-35.32, -76.2, -5) mm, rotated rx -180 ry 0 rz 90 deg; joints [71.002, -17.818, 85.279, 0, 22.54, 71.002]
  MoveC 3265 to (-31.87, -75, -5) mm, rotated rx -180 ry 0 rz 90 deg; joints [71.078, -17.765, 85.068, 0, 22.696, 71.078] to (-29.87, -71.95, -5) mm, rotated rx 180 ry 0 rz 90 deg; joints [71.197, -17.748, 85.002, 0, 22.746, 71.197]
  MoveL 3266 to (-17.27, -23.57, -5) mm, rotated rx -180 ry 0 rz 90 deg; joints [72.886, -17.803, 85.216, 0, 22.586, 72.886]
  MoveC 3267 to (-17.01, -21.98, -5) mm, rotated rx -180 ry 0 rz 90 deg; joints [72.94, -17.807, 85.233, 0, 22.574, 72.94] to (-17.06, -20.37, -5) mm, rotated rx 180 ry 0 rz 90 deg; joints [72.991, -17.816, 85.27, 0, 22.546, 72.991]
  MoveC 3268 to (-18.84, -17.28, -5) mm, rotated rx -180 ry 0 rz 90 deg; joints [73.074, -17.865, 85.461, 0, 22.404, 73.074] to (-22.27, -16.29, -5) mm, rotated rx -180 ry 0 rz 90 deg; joints [73.072, -17.931, 85.721, 0, 22.209, 73.072]
  MoveL 3269 to (-23.22, -16.41, -5) mm, rotated rx 180 ry 0 rz 90 deg; joints [73.059, -17.947, 85.785, 0, 22.162, 73.059]
  MoveL 3270 to (-27.01, -17.19, -5) mm, rotated rx 180 ry 0 rz 90 deg; joints [72.996, -18.008, 86.032, 0, 21.977, 72.996]
  MoveL 3271 to (-47.49, -21.55, -5) mm, rotated rx -180 ry 0 rz 90 deg; joints [72.646, -18.332, 87.349, 0, 20.982, 72.646]
  MoveL 3272 to (-45.92, -28.94, -5) mm, rotated rx 180 ry 0 rz 90 deg; joints [72.419, -18.267, 87.083, 0, 21.184, 72.419]
  MoveL 3273 to (-45.92, -28.94, -2) mm, rotated rx -180 ry 0 rz 90 deg; joints [72.419, -18.423, 87.184, 0, 21.238, 72.419]
  Establecer velocidad (1000.0 mm/s)
  MoveL 3274 to (-45.92, -28.94, 10) mm, rotated rx 180 ry 0 rz 90 deg; joints [72.419, -19.042, 87.583, 0, 21.459, 72.419]
  Establecer velocidad (66.7 mm/s)
  MoveL 3275 to (17.55, -67.98, 10) mm, rotated rx -180 ry 0 rz 90 deg; joints [71.825, -17.635, 82.238, 0, 25.397, 71.825]
  MoveL 3276 to (17.55, -67.98, -1.75) mm, rotated rx -180 ry 0 rz 90 deg; joints [71.825, -17.041, 81.845, 0, 25.195, 71.825]
  MoveL 3277 to (17.38, -69.49, -2.16) mm, rotated rx -180 ry 0 rz 90 deg; joints [71.776, -17.014, 81.808, 0, 25.206, 71.776]
